  PROC DrawPart91()
    MoveL Offs(pOrigin,410.01,74.28,0.00),v60,z0,tPen\WObj:=wPaper;
    MoveL Offs(pOrigin,409.38,74.91,0.00),v40,z0,tPen\WObj:=wPaper;
    MoveL Offs(pOrigin,410.01,74.28,0.00),v40,fine,tPen\WObj:=wPaper;
    MoveL Offs(pOrigin,410.01,74.28,6.00),v60,z5,tPen\WObj:=wPaper;
    MoveL Offs(pOrigin,409.80,69.81,6.00),vTravel,z5,tPen\WObj:=wPaper;
    MoveL Offs(pOrigin,409.80,69.81,0.00),v60,z0,tPen\WObj:=wPaper;
    MoveL Offs(pOrigin,407.89,71.72,0.00),v40,z0,tPen\WObj:=wPaper;
    MoveL Offs(pOrigin,409.80,69.81,0.00),v40,fine,tPen\WObj:=wPaper;
    MoveL Offs(pOrigin,409.80,69.81,6.00),v60,z5,tPen\WObj:=wPaper;
    MoveL Offs(pOrigin,410.86,68.75,6.00),vTravel,z5,tPen\WObj:=wPaper;
    MoveL Offs(pOrigin,410.86,68.75,0.00),v60,z0,tPen\WObj:=wPaper;
    MoveL Offs(pOrigin,410.23,69.39,0.00),v40,z0,tPen\WObj:=wPaper;
    MoveL Offs(pOrigin,410.86,68.75,0.00),v40,fine,tPen\WObj:=wPaper;
    MoveL Offs(pOrigin,410.86,68.75,6.00),v60,z5,tPen\WObj:=wPaper;
    MoveL Offs(pOrigin,412.49,69.10,6.00),vTravel,z5,tPen\WObj:=wPaper;
    MoveL Offs(pOrigin,412.49,69.10,0.00),v60,z0,tPen\WObj:=wPaper;
    MoveL Offs(pOrigin,409.80,71.72,0.00),v40,z0,tPen\WObj:=wPaper;
    MoveL Offs(pOrigin,412.49,69.10,0.00),v40,fine,tPen\WObj:=wPaper;
    MoveL Offs(pOrigin,412.49,69.10,6.00),v60,z5,tPen\WObj:=wPaper;
    MoveL Offs(pOrigin,412.14,67.05,6.00),vTravel,z5,tPen\WObj:=wPaper;
    MoveL Offs(pOrigin,412.14,67.05,0.00),v60,z0,tPen\WObj:=wPaper;
    MoveL Offs(pOrigin,411.29,68.11,0.00),v40,z0,tPen\WObj:=wPaper;
    MoveL Offs(pOrigin,412.14,67.05,0.00),v40,fine,tPen\WObj:=wPaper;
    MoveL Offs(pOrigin,412.14,67.05,6.00),v60,z5,tPen\WObj:=wPaper;
    MoveL Offs(pOrigin,413.20,65.35,6.00),vTravel,z5,tPen\WObj:=wPaper;
    MoveL Offs(pOrigin,413.20,65.35,0.00),v60,z0,tPen\WObj:=wPaper;
    MoveL Offs(pOrigin,412.99,65.78,0.00),v40,z0,tPen\WObj:=wPaper;
    MoveL Offs(pOrigin,413.20,65.35,0.00),v40,fine,tPen\WObj:=wPaper;
    MoveL Offs(pOrigin,413.20,65.35,6.00),v60,z5,tPen\WObj:=wPaper;
    MoveL Offs(pOrigin,409.38,62.80,6.00),vTravel,z5,tPen\WObj:=wPaper;
    MoveL Offs(pOrigin,409.38,62.80,0.00),v60,z0,tPen\WObj:=wPaper;
    MoveL Offs(pOrigin,408.81,64.50,0.00),v40,z0,tPen\WObj:=wPaper;
    MoveL Offs(pOrigin,406.97,67.69,0.00),v40,z0,tPen\WObj:=wPaper;
    MoveL Offs(pOrigin,405.62,68.54,0.00),v40,z0,tPen\WObj:=wPaper;
    MoveL Offs(pOrigin,402.79,72.36,0.00),v40,z0,tPen\WObj:=wPaper;
    MoveL Offs(pOrigin,400.66,74.28,0.00),v40,fine,tPen\WObj:=wPaper;
    MoveL Offs(pOrigin,400.66,74.28,6.00),v60,z5,tPen\WObj:=wPaper;
    MoveL Offs(pOrigin,405.55,68.32,6.00),vTravel,z5,tPen\WObj:=wPaper;
    MoveL Offs(pOrigin,405.55,68.32,0.00),v60,z0,tPen\WObj:=wPaper;
    MoveL Offs(pOrigin,405.69,67.05,0.00),v40,z0,tPen\WObj:=wPaper;
    MoveL Offs(pOrigin,407.82,62.59,0.00),v40,z0,tPen\WObj:=wPaper;
    MoveL Offs(pOrigin,409.38,56.85,0.00),v40,z0,tPen\WObj:=wPaper;
    MoveL Offs(pOrigin,409.38,56.85,0.00),v40,z0,tPen\WObj:=wPaper;
    MoveL Offs(pOrigin,410.01,56.42,0.00),v40,z0,tPen\WObj:=wPaper;
    MoveL Offs(pOrigin,409.80,55.58,0.00),v40,z0,tPen\WObj:=wPaper;
    MoveL Offs(pOrigin,409.80,55.58,0.00),v40,z0,tPen\WObj:=wPaper;
    MoveL Offs(pOrigin,410.23,54.94,0.00),v40,z0,tPen\WObj:=wPaper;
    MoveL Offs(pOrigin,410.08,53.66,0.00),v40,z0,tPen\WObj:=wPaper;
    MoveL Offs(pOrigin,410.44,53.03,0.00),v40,z0,tPen\WObj:=wPaper;
    MoveL Offs(pOrigin,410.23,49.84,0.00),v40,z0,tPen\WObj:=wPaper;
    MoveL Offs(pOrigin,410.23,49.84,0.00),v40,z0,tPen\WObj:=wPaper;
    MoveL Offs(pOrigin,410.01,48.14,0.00),v40,z0,tPen\WObj:=wPaper;
    MoveL Offs(pOrigin,410.01,48.14,0.00),v40,z0,tPen\WObj:=wPaper;
    MoveL Offs(pOrigin,409.80,46.86,0.00),v40,z0,tPen\WObj:=wPaper;
    MoveL Offs(pOrigin,409.80,46.86,0.00),v40,z0,tPen\WObj:=wPaper;
    MoveL Offs(pOrigin,409.80,46.22,0.00),v40,z0,tPen\WObj:=wPaper;
    MoveL Offs(pOrigin,409.16,45.80,0.00),v40,z0,tPen\WObj:=wPaper;
    MoveL Offs(pOrigin,409.16,45.80,0.00),v40,z0,tPen\WObj:=wPaper;
    MoveL Offs(pOrigin,408.31,42.61,0.00),v40,fine,tPen\WObj:=wPaper;
    MoveL Offs(pOrigin,408.31,42.61,6.00),v60,z5,tPen\WObj:=wPaper;
    MoveL Offs(pOrigin,409.80,43.25,6.00),vTravel,z5,tPen\WObj:=wPaper;
    MoveL Offs(pOrigin,409.80,43.25,0.00),v60,z0,tPen\WObj:=wPaper;
    MoveL Offs(pOrigin,410.23,43.67,0.00),v40,z0,tPen\WObj:=wPaper;
    MoveL Offs(pOrigin,409.80,43.25,0.00),v40,fine,tPen\WObj:=wPaper;
    MoveL Offs(pOrigin,409.80,43.25,6.00),v60,z5,tPen\WObj:=wPaper;
    MoveL Offs(pOrigin,410.86,44.31,6.00),vTravel,z5,tPen\WObj:=wPaper;
    MoveL Offs(pOrigin,410.86,44.31,0.00),v60,z0,tPen\WObj:=wPaper;
    MoveL Offs(pOrigin,411.29,44.95,0.00),v40,z0,tPen\WObj:=wPaper;
    MoveL Offs(pOrigin,410.86,44.31,0.00),v40,fine,tPen\WObj:=wPaper;
    MoveL Offs(pOrigin,410.86,44.31,6.00),v60,z5,tPen\WObj:=wPaper;
    MoveL Offs(pOrigin,412.14,43.25,6.00),vTravel,z5,tPen\WObj:=wPaper;
    MoveL Offs(pOrigin,412.14,43.25,0.00),v60,z0,tPen\WObj:=wPaper;
    MoveL Offs(pOrigin,412.56,43.67,0.00),v40,z0,tPen\WObj:=wPaper;
    MoveL Offs(pOrigin,412.14,43.25,0.00),v40,fine,tPen\WObj:=wPaper;
    MoveL Offs(pOrigin,412.14,43.25,6.00),v60,z5,tPen\WObj:=wPaper;
    MoveL Offs(pOrigin,412.99,44.31,6.00),vTravel,z5,tPen\WObj:=wPaper;
    MoveL Offs(pOrigin,412.99,44.31,0.00),v60,z0,tPen\WObj:=wPaper;
    MoveL Offs(pOrigin,413.20,44.74,0.00),v40,z0,tPen\WObj:=wPaper;
    MoveL Offs(pOrigin,412.99,44.31,0.00),v40,z0,tPen\WObj:=wPaper;
    MoveL Offs(pOrigin,413.41,44.95,0.00),v40,z0,tPen\WObj:=wPaper;
    MoveL Offs(pOrigin,413.62,45.38,0.00),v40,z0,tPen\WObj:=wPaper;
    MoveL Offs(pOrigin,413.41,44.95,0.00),v40,z0,tPen\WObj:=wPaper;
    MoveL Offs(pOrigin,413.84,45.80,0.00),v40,z0,tPen\WObj:=wPaper;
    MoveL Offs(pOrigin,414.05,46.22,0.00),v40,z0,tPen\WObj:=wPaper;
    MoveL Offs(pOrigin,413.84,45.80,0.00),v40,fine,tPen\WObj:=wPaper;
    MoveL Offs(pOrigin,413.84,45.80,6.00),v60,z5,tPen\WObj:=wPaper;
    MoveL Offs(pOrigin,412.35,46.86,6.00),vTravel,z5,tPen\WObj:=wPaper;
    MoveL Offs(pOrigin,412.35,46.86,0.00),v60,z0,tPen\WObj:=wPaper;
    MoveL Offs(pOrigin,412.56,47.29,0.00),v40,z0,tPen\WObj:=wPaper;
    MoveL Offs(pOrigin,412.35,46.86,0.00),v40,fine,tPen\WObj:=wPaper;
    MoveL Offs(pOrigin,412.35,46.86,6.00),v60,z5,tPen\WObj:=wPaper;
    MoveL Offs(pOrigin,409.16,46.86,6.00),vTravel,z5,tPen\WObj:=wPaper;
    MoveL Offs(pOrigin,409.16,46.86,0.00),v60,z0,tPen\WObj:=wPaper;
    MoveL Offs(pOrigin,408.95,46.01,0.00),v40,z0,tPen\WObj:=wPaper;
    MoveL Offs(pOrigin,409.16,45.80,0.00),v40,z0,tPen\WObj:=wPaper;
    MoveL Offs(pOrigin,409.16,46.86,0.00),v40,z0,tPen\WObj:=wPaper;
    MoveL Offs(pOrigin,409.38,48.14,0.00),v40,z0,tPen\WObj:=wPaper;
    MoveL Offs(pOrigin,409.38,48.14,0.00),v40,z0,tPen\WObj:=wPaper;
    MoveL Offs(pOrigin,409.59,49.84,0.00),v40,z0,tPen\WObj:=wPaper;
    MoveL Offs(pOrigin,409.59,49.84,0.00),v40,z0,tPen\WObj:=wPaper;
    MoveL Offs(pOrigin,409.80,53.66,0.00),v40,z0,tPen\WObj:=wPaper;
    MoveL Offs(pOrigin,410.01,54.09,0.00),v40,z0,tPen\WObj:=wPaper;
    MoveL Offs(pOrigin,409.80,53.88,0.00),v40,z0,tPen\WObj:=wPaper;
    MoveL Offs(pOrigin,409.38,54.30,0.00),v40,z0,tPen\WObj:=wPaper;
    MoveL Offs(pOrigin,409.38,55.36,0.00),v40,z0,tPen\WObj:=wPaper;
    MoveL Offs(pOrigin,409.80,55.58,0.00),v40,z0,tPen\WObj:=wPaper;
    MoveL Offs(pOrigin,409.38,55.58,0.00),v40,z0,tPen\WObj:=wPaper;
    MoveL Offs(pOrigin,409.16,56.64,0.00),v40,z0,tPen\WObj:=wPaper;
    MoveL Offs(pOrigin,409.38,56.85,0.00),v40,fine,tPen\WObj:=wPaper;
    MoveL Offs(pOrigin,409.38,56.85,6.00),v60,z5,tPen\WObj:=wPaper;
    MoveL Offs(pOrigin,407.04,64.07,6.00),vTravel,z5,tPen\WObj:=wPaper;
    MoveL Offs(pOrigin,407.04,64.07,0.00),v60,z0,tPen\WObj:=wPaper;
    MoveL Offs(pOrigin,406.83,64.50,0.00),v40,z0,tPen\WObj:=wPaper;
    MoveL Offs(pOrigin,407.04,64.07,0.00),v40,fine,tPen\WObj:=wPaper;
    MoveL Offs(pOrigin,407.04,64.07,6.00),v60,z5,tPen\WObj:=wPaper;
    MoveL Offs(pOrigin,397.69,57.49,6.00),vTravel,z5,tPen\WObj:=wPaper;
    MoveL Offs(pOrigin,397.69,57.49,0.00),v60,z0,tPen\WObj:=wPaper;
    MoveL Offs(pOrigin,397.26,58.12,0.00),v40,z0,tPen\WObj:=wPaper;
    MoveL Offs(pOrigin,397.69,57.49,0.00),v40,fine,tPen\WObj:=wPaper;
    MoveL Offs(pOrigin,397.69,57.49,6.00),v60,z5,tPen\WObj:=wPaper;
  ENDPROC

  PROC DrawPart92()
    MoveL Offs(pOrigin,398.33,56.42,6.00),vTravel,z5,tPen\WObj:=wPaper;
    MoveL Offs(pOrigin,398.33,56.42,0.00),v60,z0,tPen\WObj:=wPaper;
    MoveL Offs(pOrigin,398.11,56.85,0.00),v40,z0,tPen\WObj:=wPaper;
    MoveL Offs(pOrigin,398.33,56.42,0.00),v40,fine,tPen\WObj:=wPaper;
    MoveL Offs(pOrigin,398.33,56.42,6.00),v60,z5,tPen\WObj:=wPaper;
    MoveL Offs(pOrigin,396.84,58.76,6.00),vTravel,z5,tPen\WObj:=wPaper;
    MoveL Offs(pOrigin,396.84,58.76,0.00),v60,z0,tPen\WObj:=wPaper;
    MoveL Offs(pOrigin,396.41,59.40,0.00),v40,z0,tPen\WObj:=wPaper;
    MoveL Offs(pOrigin,396.84,58.76,0.00),v40,fine,tPen\WObj:=wPaper;
    MoveL Offs(pOrigin,396.84,58.76,6.00),v60,z5,tPen\WObj:=wPaper;
    MoveL Offs(pOrigin,395.56,60.67,6.00),vTravel,z5,tPen\WObj:=wPaper;
    MoveL Offs(pOrigin,395.56,60.67,0.00),v60,z0,tPen\WObj:=wPaper;
    MoveL Offs(pOrigin,395.14,61.10,0.00),v40,z0,tPen\WObj:=wPaper;
    MoveL Offs(pOrigin,395.56,60.67,0.00),v40,fine,tPen\WObj:=wPaper;
    MoveL Offs(pOrigin,395.56,60.67,6.00),v60,z5,tPen\WObj:=wPaper;
    MoveL Offs(pOrigin,394.29,62.16,6.00),vTravel,z5,tPen\WObj:=wPaper;
    MoveL Offs(pOrigin,394.29,62.16,0.00),v60,z0,tPen\WObj:=wPaper;
    MoveL Offs(pOrigin,393.86,62.80,0.00),v40,z0,tPen\WObj:=wPaper;
    MoveL Offs(pOrigin,394.29,62.16,0.00),v40,fine,tPen\WObj:=wPaper;
    MoveL Offs(pOrigin,394.29,62.16,6.00),v60,z5,tPen\WObj:=wPaper;
    MoveL Offs(pOrigin,393.44,63.22,6.00),vTravel,z5,tPen\WObj:=wPaper;
    MoveL Offs(pOrigin,393.44,63.22,0.00),v60,z0,tPen\WObj:=wPaper;
    MoveL Offs(pOrigin,393.01,63.65,0.00),v40,z0,tPen\WObj:=wPaper;
    MoveL Offs(pOrigin,393.44,63.22,0.00),v40,fine,tPen\WObj:=wPaper;
    MoveL Offs(pOrigin,393.44,63.22,6.00),v60,z5,tPen\WObj:=wPaper;
    MoveL Offs(pOrigin,392.16,64.71,6.00),vTravel,z5,tPen\WObj:=wPaper;
    MoveL Offs(pOrigin,392.16,64.71,0.00),v60,z0,tPen\WObj:=wPaper;
    MoveL Offs(pOrigin,391.52,65.35,0.00),v40,z0,tPen\WObj:=wPaper;
    MoveL Offs(pOrigin,392.16,64.71,0.00),v40,fine,tPen\WObj:=wPaper;
    MoveL Offs(pOrigin,392.16,64.71,6.00),v60,z5,tPen\WObj:=wPaper;
    MoveL Offs(pOrigin,391.31,65.56,6.00),vTravel,z5,tPen\WObj:=wPaper;
    MoveL Offs(pOrigin,391.31,65.56,0.00),v60,z0,tPen\WObj:=wPaper;
    MoveL Offs(pOrigin,390.67,66.20,0.00),v40,z0,tPen\WObj:=wPaper;
    MoveL Offs(pOrigin,391.31,65.56,0.00),v40,fine,tPen\WObj:=wPaper;
    MoveL Offs(pOrigin,391.31,65.56,6.00),v60,z5,tPen\WObj:=wPaper;
    MoveL Offs(pOrigin,389.61,67.05,6.00),vTravel,z5,tPen\WObj:=wPaper;
    MoveL Offs(pOrigin,389.61,67.05,0.00),v60,z0,tPen\WObj:=wPaper;
    MoveL Offs(pOrigin,388.98,67.69,0.00),v40,z0,tPen\WObj:=wPaper;
    MoveL Offs(pOrigin,389.61,67.05,0.00),v40,fine,tPen\WObj:=wPaper;
    MoveL Offs(pOrigin,389.61,67.05,6.00),v60,z5,tPen\WObj:=wPaper;
    MoveL Offs(pOrigin,399.81,53.66,6.00),vTravel,z5,tPen\WObj:=wPaper;
    MoveL Offs(pOrigin,399.81,53.66,0.00),v60,z0,tPen\WObj:=wPaper;
    MoveL Offs(pOrigin,399.60,54.09,0.00),v40,z0,tPen\WObj:=wPaper;
    MoveL Offs(pOrigin,399.81,53.66,0.00),v40,fine,tPen\WObj:=wPaper;
    MoveL Offs(pOrigin,399.81,53.66,6.00),v60,z5,tPen\WObj:=wPaper;
    MoveL Offs(pOrigin,402.58,42.19,6.00),vTravel,z5,tPen\WObj:=wPaper;
    MoveL Offs(pOrigin,402.58,42.19,0.00),v60,z0,tPen\WObj:=wPaper;
    MoveL Offs(pOrigin,401.94,47.71,0.00),v40,z0,tPen\WObj:=wPaper;
    MoveL Offs(pOrigin,399.88,53.88,0.00),v40,z0,tPen\WObj:=wPaper;
    MoveL Offs(pOrigin,396.20,60.04,0.00),v40,z0,tPen\WObj:=wPaper;
    MoveL Offs(pOrigin,392.59,64.50,0.00),v40,z0,tPen\WObj:=wPaper;
    MoveL Offs(pOrigin,387.91,68.75,0.00),v40,z0,tPen\WObj:=wPaper;
    MoveL Offs(pOrigin,382.81,72.22,0.00),v40,z0,tPen\WObj:=wPaper;
    MoveL Offs(pOrigin,377.08,74.77,0.00),v40,z0,tPen\WObj:=wPaper;
    MoveL Offs(pOrigin,370.49,76.40,0.00),v40,z0,tPen\WObj:=wPaper;
    MoveL Offs(pOrigin,370.42,76.19,0.00),v40,z0,tPen\WObj:=wPaper;
    MoveL Offs(pOrigin,369.64,75.97,0.00),v40,z0,tPen\WObj:=wPaper;
    MoveL Offs(pOrigin,369.00,76.61,0.00),v40,z0,tPen\WObj:=wPaper;
    MoveL Offs(pOrigin,369.85,76.82,0.00),v40,z0,tPen\WObj:=wPaper;
    MoveL Offs(pOrigin,370.42,76.19,0.00),v40,fine,tPen\WObj:=wPaper;
    MoveL Offs(pOrigin,370.42,76.19,6.00),v60,z5,tPen\WObj:=wPaper;
    MoveL Offs(pOrigin,381.96,113.38,6.00),vTravel,z5,tPen\WObj:=wPaper;
    MoveL Offs(pOrigin,381.96,113.38,0.00),v60,z0,tPen\WObj:=wPaper;
    MoveL Offs(pOrigin,386.42,112.74,0.00),v40,z0,tPen\WObj:=wPaper;
    MoveL Offs(pOrigin,391.10,111.46,0.00),v40,z0,tPen\WObj:=wPaper;
    MoveL Offs(pOrigin,391.10,111.46,0.00),v40,z0,tPen\WObj:=wPaper;
    MoveL Offs(pOrigin,393.86,110.68,0.00),v40,z0,tPen\WObj:=wPaper;
    MoveL Offs(pOrigin,399.17,107.71,0.00),v40,z0,tPen\WObj:=wPaper;
    MoveL Offs(pOrigin,399.95,107.64,0.00),v40,z0,tPen\WObj:=wPaper;
    MoveL Offs(pOrigin,400.02,108.28,0.00),v40,z0,tPen\WObj:=wPaper;
    MoveL Offs(pOrigin,398.61,112.53,0.00),v40,z0,tPen\WObj:=wPaper;
    MoveL Offs(pOrigin,396.06,116.21,0.00),v40,z0,tPen\WObj:=wPaper;
    MoveL Offs(pOrigin,395.14,118.47,0.00),v40,z0,tPen\WObj:=wPaper;
    MoveL Offs(pOrigin,395.35,125.06,0.00),v40,z0,tPen\WObj:=wPaper;
    MoveL Offs(pOrigin,395.00,126.12,0.00),v40,z0,tPen\WObj:=wPaper;
    MoveL Offs(pOrigin,393.65,126.97,0.00),v40,z0,tPen\WObj:=wPaper;
    MoveL Offs(pOrigin,392.16,126.97,0.00),v40,z0,tPen\WObj:=wPaper;
    MoveL Offs(pOrigin,385.36,125.49,0.00),v40,z0,tPen\WObj:=wPaper;
    MoveL Offs(pOrigin,384.51,125.70,0.00),v40,z0,tPen\WObj:=wPaper;
    MoveL Offs(pOrigin,384.51,125.70,0.00),v40,z0,tPen\WObj:=wPaper;
    MoveL Offs(pOrigin,378.99,124.64,0.00),v40,fine,tPen\WObj:=wPaper;
    MoveL Offs(pOrigin,378.99,124.64,6.00),v60,z5,tPen\WObj:=wPaper;
    MoveL Offs(pOrigin,394.71,126.34,6.00),vTravel,z5,tPen\WObj:=wPaper;
    MoveL Offs(pOrigin,394.71,126.34,0.00),v60,z0,tPen\WObj:=wPaper;
    MoveL Offs(pOrigin,394.50,126.76,0.00),v40,z0,tPen\WObj:=wPaper;
    MoveL Offs(pOrigin,394.71,126.34,0.00),v40,fine,tPen\WObj:=wPaper;
    MoveL Offs(pOrigin,394.71,126.34,6.00),v60,z5,tPen\WObj:=wPaper;
    MoveL Offs(pOrigin,396.41,126.55,6.00),vTravel,z5,tPen\WObj:=wPaper;
    MoveL Offs(pOrigin,396.41,126.55,0.00),v60,z0,tPen\WObj:=wPaper;
    MoveL Offs(pOrigin,396.20,126.97,0.00),v40,z0,tPen\WObj:=wPaper;
    MoveL Offs(pOrigin,396.41,126.55,0.00),v40,fine,tPen\WObj:=wPaper;
    MoveL Offs(pOrigin,396.41,126.55,6.00),v60,z5,tPen\WObj:=wPaper;
    MoveL Offs(pOrigin,397.26,117.20,6.00),vTravel,z5,tPen\WObj:=wPaper;
    MoveL Offs(pOrigin,397.26,117.20,0.00),v60,z0,tPen\WObj:=wPaper;
    MoveL Offs(pOrigin,397.05,117.62,0.00),v40,z0,tPen\WObj:=wPaper;
    MoveL Offs(pOrigin,397.26,117.20,0.00),v40,fine,tPen\WObj:=wPaper;
    MoveL Offs(pOrigin,397.26,117.20,6.00),v60,z5,tPen\WObj:=wPaper;
    MoveL Offs(pOrigin,398.11,116.14,6.00),vTravel,z5,tPen\WObj:=wPaper;
    MoveL Offs(pOrigin,398.11,116.14,0.00),v60,z0,tPen\WObj:=wPaper;
    MoveL Offs(pOrigin,398.33,115.71,0.00),v40,z0,tPen\WObj:=wPaper;
    MoveL Offs(pOrigin,398.11,116.14,0.00),v40,fine,tPen\WObj:=wPaper;
    MoveL Offs(pOrigin,398.11,116.14,6.00),v60,z5,tPen\WObj:=wPaper;
    MoveL Offs(pOrigin,396.84,115.07,6.00),vTravel,z5,tPen\WObj:=wPaper;
    MoveL Offs(pOrigin,396.84,115.07,0.00),v60,z0,tPen\WObj:=wPaper;
    MoveL Offs(pOrigin,396.62,115.50,0.00),v40,z0,tPen\WObj:=wPaper;
    MoveL Offs(pOrigin,396.84,115.07,0.00),v40,fine,tPen\WObj:=wPaper;
    MoveL Offs(pOrigin,396.84,115.07,6.00),v60,z5,tPen\WObj:=wPaper;
    MoveL Offs(pOrigin,399.81,113.38,6.00),vTravel,z5,tPen\WObj:=wPaper;
    MoveL Offs(pOrigin,399.81,113.38,0.00),v60,z0,tPen\WObj:=wPaper;
    MoveL Offs(pOrigin,399.60,113.80,0.00),v40,z0,tPen\WObj:=wPaper;
    MoveL Offs(pOrigin,399.81,113.38,0.00),v40,fine,tPen\WObj:=wPaper;
    MoveL Offs(pOrigin,399.81,113.38,6.00),v60,z5,tPen\WObj:=wPaper;
    MoveL Offs(pOrigin,398.11,106.79,6.00),vTravel,z5,tPen\WObj:=wPaper;
    MoveL Offs(pOrigin,398.11,106.79,0.00),v60,z0,tPen\WObj:=wPaper;
    MoveL Offs(pOrigin,398.40,106.65,0.00),v40,z0,tPen\WObj:=wPaper;
    MoveL Offs(pOrigin,395.35,108.77,0.00),v40,z0,tPen\WObj:=wPaper;
    MoveL Offs(pOrigin,391.74,110.54,0.00),v40,z0,tPen\WObj:=wPaper;
    MoveL Offs(pOrigin,391.10,111.46,0.00),v40,fine,tPen\WObj:=wPaper;
    MoveL Offs(pOrigin,391.10,111.46,6.00),v60,z5,tPen\WObj:=wPaper;
    MoveL Offs(pOrigin,403.21,104.24,6.00),vTravel,z5,tPen\WObj:=wPaper;
  ENDPROC

  PROC DrawPart93()
    MoveL Offs(pOrigin,403.21,104.24,0.00),v60,z0,tPen\WObj:=wPaper;
    MoveL Offs(pOrigin,403.00,104.66,0.00),v40,z0,tPen\WObj:=wPaper;
    MoveL Offs(pOrigin,403.21,104.24,0.00),v40,z0,tPen\WObj:=wPaper;
    MoveL Offs(pOrigin,403.85,103.60,0.00),v40,z0,tPen\WObj:=wPaper;
    MoveL Offs(pOrigin,403.64,104.03,0.00),v40,z0,tPen\WObj:=wPaper;
    MoveL Offs(pOrigin,403.85,103.60,0.00),v40,fine,tPen\WObj:=wPaper;
    MoveL Offs(pOrigin,403.85,103.60,6.00),v60,z5,tPen\WObj:=wPaper;
    MoveL Offs(pOrigin,385.58,153.32,6.00),vTravel,z5,tPen\WObj:=wPaper;
    MoveL Offs(pOrigin,385.58,153.32,0.00),v60,z0,tPen\WObj:=wPaper;
    MoveL Offs(pOrigin,385.36,153.75,0.00),v40,z0,tPen\WObj:=wPaper;
    MoveL Offs(pOrigin,385.58,153.32,0.00),v40,fine,tPen\WObj:=wPaper;
    MoveL Offs(pOrigin,385.58,153.32,6.00),v60,z5,tPen\WObj:=wPaper;
    MoveL Offs(pOrigin,383.88,153.11,6.00),vTravel,z5,tPen\WObj:=wPaper;
    MoveL Offs(pOrigin,383.88,153.11,0.00),v60,z0,tPen\WObj:=wPaper;
    MoveL Offs(pOrigin,383.66,153.54,0.00),v40,z0,tPen\WObj:=wPaper;
    MoveL Offs(pOrigin,383.88,153.11,0.00),v40,fine,tPen\WObj:=wPaper;
    MoveL Offs(pOrigin,383.88,153.11,6.00),v60,z5,tPen\WObj:=wPaper;
    MoveL Offs(pOrigin,383.24,154.60,6.00),vTravel,z5,tPen\WObj:=wPaper;
    MoveL Offs(pOrigin,383.24,154.60,0.00),v60,z0,tPen\WObj:=wPaper;
    MoveL Offs(pOrigin,383.02,155.02,0.00),v40,z0,tPen\WObj:=wPaper;
    MoveL Offs(pOrigin,383.24,154.60,0.00),v40,z0,tPen\WObj:=wPaper;
    MoveL Offs(pOrigin,382.81,155.45,0.00),v40,z0,tPen\WObj:=wPaper;
    MoveL Offs(pOrigin,382.60,155.88,0.00),v40,z0,tPen\WObj:=wPaper;
    MoveL Offs(pOrigin,382.81,155.45,0.00),v40,z0,tPen\WObj:=wPaper;
    MoveL Offs(pOrigin,382.39,156.30,0.00),v40,z0,tPen\WObj:=wPaper;
    MoveL Offs(pOrigin,382.17,156.73,0.00),v40,z0,tPen\WObj:=wPaper;
    MoveL Offs(pOrigin,382.39,156.30,0.00),v40,fine,tPen\WObj:=wPaper;
    MoveL Offs(pOrigin,382.39,156.30,6.00),v60,z5,tPen\WObj:=wPaper;
    MoveL Offs(pOrigin,381.75,157.57,6.00),vTravel,z5,tPen\WObj:=wPaper;
    MoveL Offs(pOrigin,381.75,157.57,0.00),v60,z0,tPen\WObj:=wPaper;
    MoveL Offs(pOrigin,381.54,158.00,0.00),v40,z0,tPen\WObj:=wPaper;
    MoveL Offs(pOrigin,381.75,157.57,0.00),v40,fine,tPen\WObj:=wPaper;
    MoveL Offs(pOrigin,381.75,157.57,6.00),v60,z5,tPen\WObj:=wPaper;
    MoveL Offs(pOrigin,383.02,158.64,6.00),vTravel,z5,tPen\WObj:=wPaper;
    MoveL Offs(pOrigin,383.02,158.64,0.00),v60,z0,tPen\WObj:=wPaper;
    MoveL Offs(pOrigin,382.81,159.06,0.00),v40,z0,tPen\WObj:=wPaper;
    MoveL Offs(pOrigin,383.02,158.64,0.00),v40,z0,tPen\WObj:=wPaper;
    MoveL Offs(pOrigin,383.45,157.79,0.00),v40,z0,tPen\WObj:=wPaper;
    MoveL Offs(pOrigin,383.24,158.21,0.00),v40,z0,tPen\WObj:=wPaper;
    MoveL Offs(pOrigin,383.45,157.79,0.00),v40,fine,tPen\WObj:=wPaper;
    MoveL Offs(pOrigin,383.45,157.79,6.00),v60,z5,tPen\WObj:=wPaper;
    MoveL Offs(pOrigin,384.51,155.66,6.00),vTravel,z5,tPen\WObj:=wPaper;
    MoveL Offs(pOrigin,384.51,155.66,0.00),v60,z0,tPen\WObj:=wPaper;
    MoveL Offs(pOrigin,384.30,156.09,0.00),v40,z0,tPen\WObj:=wPaper;
    MoveL Offs(pOrigin,384.51,155.66,0.00),v40,fine,tPen\WObj:=wPaper;
    MoveL Offs(pOrigin,384.51,155.66,6.00),v60,z5,tPen\WObj:=wPaper;
    MoveL Offs(pOrigin,369.42,186.48,6.00),vTravel,z5,tPen\WObj:=wPaper;
    MoveL Offs(pOrigin,369.42,186.48,0.00),v60,z0,tPen\WObj:=wPaper;
    MoveL Offs(pOrigin,369.64,186.90,0.00),v40,z0,tPen\WObj:=wPaper;
    MoveL Offs(pOrigin,369.42,186.48,0.00),v40,fine,tPen\WObj:=wPaper;
    MoveL Offs(pOrigin,369.42,186.48,6.00),v60,z5,tPen\WObj:=wPaper;
    MoveL Offs(pOrigin,368.58,187.75,6.00),vTravel,z5,tPen\WObj:=wPaper;
    MoveL Offs(pOrigin,368.58,187.75,0.00),v60,z0,tPen\WObj:=wPaper;
    MoveL Offs(pOrigin,369.00,188.18,0.00),v40,z0,tPen\WObj:=wPaper;
    MoveL Offs(pOrigin,368.58,187.75,0.00),v40,fine,tPen\WObj:=wPaper;
    MoveL Offs(pOrigin,368.58,187.75,6.00),v60,z5,tPen\WObj:=wPaper;
    MoveL Offs(pOrigin,367.73,186.26,6.00),vTravel,z5,tPen\WObj:=wPaper;
    MoveL Offs(pOrigin,367.73,186.26,0.00),v60,z0,tPen\WObj:=wPaper;
    MoveL Offs(pOrigin,367.94,186.69,0.00),v40,z0,tPen\WObj:=wPaper;
    MoveL Offs(pOrigin,367.73,186.26,0.00),v40,fine,tPen\WObj:=wPaper;
    MoveL Offs(pOrigin,367.73,186.26,6.00),v60,z5,tPen\WObj:=wPaper;
    MoveL Offs(pOrigin,341.80,182.01,6.00),vTravel,z5,tPen\WObj:=wPaper;
    MoveL Offs(pOrigin,341.80,182.01,0.00),v60,z0,tPen\WObj:=wPaper;
    MoveL Offs(pOrigin,334.15,175.85,0.00),v40,z0,tPen\WObj:=wPaper;
    MoveL Offs(pOrigin,330.33,172.02,0.00),v40,z0,tPen\WObj:=wPaper;
    MoveL Offs(pOrigin,323.74,164.16,0.00),v40,z0,tPen\WObj:=wPaper;
    MoveL Offs(pOrigin,315.38,151.84,0.00),v40,z0,tPen\WObj:=wPaper;
    MoveL Offs(pOrigin,309.85,141.64,0.00),v40,z0,tPen\WObj:=wPaper;
    MoveL Offs(pOrigin,309.08,139.51,0.00),v40,fine,tPen\WObj:=wPaper;
    MoveL Offs(pOrigin,309.08,139.51,6.00),v60,z5,tPen\WObj:=wPaper;
    MoveL Offs(pOrigin,316.73,153.75,6.00),vTravel,z5,tPen\WObj:=wPaper;
    MoveL Offs(pOrigin,316.73,153.75,0.00),v60,z0,tPen\WObj:=wPaper;
    MoveL Offs(pOrigin,316.94,154.18,0.00),v40,z0,tPen\WObj:=wPaper;
    MoveL Offs(pOrigin,316.73,153.75,0.00),v40,z0,tPen\WObj:=wPaper;
    MoveL Offs(pOrigin,317.15,154.39,0.00),v40,z0,tPen\WObj:=wPaper;
    MoveL Offs(pOrigin,317.36,154.81,0.00),v40,z0,tPen\WObj:=wPaper;
    MoveL Offs(pOrigin,317.15,154.39,0.00),v40,fine,tPen\WObj:=wPaper;
    MoveL Offs(pOrigin,317.15,154.39,6.00),v60,z5,tPen\WObj:=wPaper;
    MoveL Offs(pOrigin,305.25,169.69,6.00),vTravel,z5,tPen\WObj:=wPaper;
    MoveL Offs(pOrigin,305.25,169.69,0.00),v60,z0,tPen\WObj:=wPaper;
    MoveL Offs(pOrigin,295.90,173.09,0.00),v40,fine,tPen\WObj:=wPaper;
    MoveL Offs(pOrigin,295.90,173.09,6.00),v60,z5,tPen\WObj:=wPaper;
    MoveL Offs(pOrigin,276.56,176.70,6.00),vTravel,z5,tPen\WObj:=wPaper;
    MoveL Offs(pOrigin,276.56,176.70,0.00),v60,z0,tPen\WObj:=wPaper;
    MoveL Offs(pOrigin,276.00,174.36,0.00),v40,z0,tPen\WObj:=wPaper;
    MoveL Offs(pOrigin,271.82,165.44,0.00),v40,z0,tPen\WObj:=wPaper;
    MoveL Offs(pOrigin,268.70,157.15,0.00),v40,fine,tPen\WObj:=wPaper;
    MoveL Offs(pOrigin,268.70,157.15,6.00),v60,z5,tPen\WObj:=wPaper;
    MoveL Offs(pOrigin,274.44,150.56,6.00),vTravel,z5,tPen\WObj:=wPaper;
    MoveL Offs(pOrigin,274.44,150.56,0.00),v60,z0,tPen\WObj:=wPaper;
    MoveL Offs(pOrigin,273.73,149.93,0.00),v40,z0,tPen\WObj:=wPaper;
    MoveL Offs(pOrigin,267.78,135.05,0.00),v40,z0,tPen\WObj:=wPaper;
    MoveL Offs(pOrigin,267.64,133.77,0.00),v40,fine,tPen\WObj:=wPaper;
    MoveL Offs(pOrigin,267.64,133.77,6.00),v60,z5,tPen\WObj:=wPaper;
    MoveL Offs(pOrigin,276.14,186.48,6.00),vTravel,z5,tPen\WObj:=wPaper;
    MoveL Offs(pOrigin,276.14,186.48,0.00),v60,z0,tPen\WObj:=wPaper;
    MoveL Offs(pOrigin,275.71,187.11,0.00),v40,z0,tPen\WObj:=wPaper;
    MoveL Offs(pOrigin,276.14,186.48,0.00),v40,fine,tPen\WObj:=wPaper;
    MoveL Offs(pOrigin,276.14,186.48,6.00),v60,z5,tPen\WObj:=wPaper;
    MoveL Offs(pOrigin,303.55,208.15,6.00),vTravel,z5,tPen\WObj:=wPaper;
    MoveL Offs(pOrigin,303.55,208.15,0.00),v60,z0,tPen\WObj:=wPaper;
    MoveL Offs(pOrigin,303.12,208.79,0.00),v40,z0,tPen\WObj:=wPaper;
    MoveL Offs(pOrigin,303.55,208.15,0.00),v40,fine,tPen\WObj:=wPaper;
    MoveL Offs(pOrigin,303.55,208.15,6.00),v60,z5,tPen\WObj:=wPaper;
    MoveL Offs(pOrigin,304.40,207.30,6.00),vTravel,z5,tPen\WObj:=wPaper;
    MoveL Offs(pOrigin,304.40,207.30,0.00),v60,z0,tPen\WObj:=wPaper;
    MoveL Offs(pOrigin,303.76,207.94,0.00),v40,z0,tPen\WObj:=wPaper;
    MoveL Offs(pOrigin,304.40,207.30,0.00),v40,fine,tPen\WObj:=wPaper;
    MoveL Offs(pOrigin,304.40,207.30,6.00),v60,z5,tPen\WObj:=wPaper;
    MoveL Offs(pOrigin,314.60,193.91,6.00),vTravel,z5,tPen\WObj:=wPaper;
    MoveL Offs(pOrigin,314.60,193.91,0.00),v60,z0,tPen\WObj:=wPaper;
    MoveL Offs(pOrigin,315.02,194.12,0.00),v40,z0,tPen\WObj:=wPaper;
    MoveL Offs(pOrigin,314.60,193.91,0.00),v40,fine,tPen\WObj:=wPaper;
    MoveL Offs(pOrigin,314.60,193.91,6.00),v60,z5,tPen\WObj:=wPaper;
    MoveL Offs(pOrigin,332.66,174.15,6.00),vTravel,z5,tPen\WObj:=wPaper;
    MoveL Offs(pOrigin,332.66,174.15,0.00),v60,z0,tPen\WObj:=wPaper;
    MoveL Offs(pOrigin,333.51,175.00,0.00),v40,z0,tPen\WObj:=wPaper;
    MoveL Offs(pOrigin,332.66,174.15,0.00),v40,fine,tPen\WObj:=wPaper;
    MoveL Offs(pOrigin,332.66,174.15,6.00),v60,z5,tPen\WObj:=wPaper;
    MoveL Offs(pOrigin,331.17,172.66,6.00),vTravel,z5,tPen\WObj:=wPaper;
  ENDPROC

  PROC DrawPart94()
    MoveL Offs(pOrigin,331.17,172.66,0.00),v60,z0,tPen\WObj:=wPaper;
    MoveL Offs(pOrigin,332.02,173.51,0.00),v40,z0,tPen\WObj:=wPaper;
    MoveL Offs(pOrigin,331.17,172.66,0.00),v40,fine,tPen\WObj:=wPaper;
    MoveL Offs(pOrigin,331.17,172.66,6.00),v60,z5,tPen\WObj:=wPaper;
    MoveL Offs(pOrigin,383.66,227.27,6.00),vTravel,z5,tPen\WObj:=wPaper;
    MoveL Offs(pOrigin,383.66,227.27,0.00),v60,z0,tPen\WObj:=wPaper;
    MoveL Offs(pOrigin,383.45,227.70,0.00),v40,z0,tPen\WObj:=wPaper;
    MoveL Offs(pOrigin,383.66,227.27,0.00),v40,fine,tPen\WObj:=wPaper;
    MoveL Offs(pOrigin,383.66,227.27,6.00),v60,z5,tPen\WObj:=wPaper;
    MoveL Offs(pOrigin,250.85,225.57,6.00),vTravel,z5,tPen\WObj:=wPaper;
    MoveL Offs(pOrigin,250.85,225.57,0.00),v60,z0,tPen\WObj:=wPaper;
    MoveL Offs(pOrigin,245.54,225.15,0.00),v40,z0,tPen\WObj:=wPaper;
    MoveL Offs(pOrigin,242.56,224.30,0.00),v40,fine,tPen\WObj:=wPaper;
    MoveL Offs(pOrigin,242.56,224.30,6.00),v60,z5,tPen\WObj:=wPaper;
    MoveL Offs(pOrigin,232.15,237.05,6.00),vTravel,z5,tPen\WObj:=wPaper;
    MoveL Offs(pOrigin,232.15,237.05,0.00),v60,z0,tPen\WObj:=wPaper;
    MoveL Offs(pOrigin,232.57,237.26,0.00),v40,z0,tPen\WObj:=wPaper;
    MoveL Offs(pOrigin,232.57,238.11,0.00),v40,z0,tPen\WObj:=wPaper;
    MoveL Offs(pOrigin,231.73,238.11,0.00),v40,z0,tPen\WObj:=wPaper;
    MoveL Offs(pOrigin,231.94,238.96,0.00),v40,z0,tPen\WObj:=wPaper;
    MoveL Offs(pOrigin,233.00,239.18,0.00),v40,z0,tPen\WObj:=wPaper;
    MoveL Offs(pOrigin,233.43,238.75,0.00),v40,z0,tPen\WObj:=wPaper;
    MoveL Offs(pOrigin,233.43,238.11,0.00),v40,z0,tPen\WObj:=wPaper;
    MoveL Offs(pOrigin,233.64,238.68,0.00),v40,z0,tPen\WObj:=wPaper;
    MoveL Offs(pOrigin,235.34,239.39,0.00),v40,z0,tPen\WObj:=wPaper;
    MoveL Offs(pOrigin,235.76,240.45,0.00),v40,z0,tPen\WObj:=wPaper;
    MoveL Offs(pOrigin,235.76,240.45,0.00),v40,z0,tPen\WObj:=wPaper;
    MoveL Offs(pOrigin,234.70,240.88,0.00),v40,z0,tPen\WObj:=wPaper;
    MoveL Offs(pOrigin,234.49,241.51,0.00),v40,fine,tPen\WObj:=wPaper;
    MoveL Offs(pOrigin,234.49,241.51,6.00),v60,z5,tPen\WObj:=wPaper;
    MoveL Offs(pOrigin,238.10,242.36,6.00),vTravel,z5,tPen\WObj:=wPaper;
    MoveL Offs(pOrigin,238.10,242.36,0.00),v60,z0,tPen\WObj:=wPaper;
    MoveL Offs(pOrigin,238.31,241.94,0.00),v40,z0,tPen\WObj:=wPaper;
    MoveL Offs(pOrigin,239.16,241.73,0.00),v40,fine,tPen\WObj:=wPaper;
    MoveL Offs(pOrigin,239.16,241.73,6.00),v60,z5,tPen\WObj:=wPaper;
    MoveL Offs(pOrigin,238.10,242.36,6.00),vTravel,z5,tPen\WObj:=wPaper;
    MoveL Offs(pOrigin,238.10,242.36,0.00),v60,z0,tPen\WObj:=wPaper;
    MoveL Offs(pOrigin,236.19,242.57,0.00),v40,z0,tPen\WObj:=wPaper;
    MoveL Offs(pOrigin,233.85,241.58,0.00),v40,z0,tPen\WObj:=wPaper;
    MoveL Offs(pOrigin,232.43,243.00,0.00),v40,z0,tPen\WObj:=wPaper;
    MoveL Offs(pOrigin,231.73,246.19,0.00),v40,fine,tPen\WObj:=wPaper;
    MoveL Offs(pOrigin,231.73,246.19,6.00),v60,z5,tPen\WObj:=wPaper;
    MoveL Offs(pOrigin,231.09,237.90,6.00),vTravel,z5,tPen\WObj:=wPaper;
    MoveL Offs(pOrigin,231.09,237.90,0.00),v60,z0,tPen\WObj:=wPaper;
    MoveL Offs(pOrigin,232.15,237.05,0.00),v40,fine,tPen\WObj:=wPaper;
    MoveL Offs(pOrigin,232.15,237.05,6.00),v60,z5,tPen\WObj:=wPaper;
    MoveL Offs(pOrigin,216.43,210.91,6.00),vTravel,z5,tPen\WObj:=wPaper;
    MoveL Offs(pOrigin,216.43,210.91,0.00),v60,z0,tPen\WObj:=wPaper;
    MoveL Offs(pOrigin,217.27,211.76,0.00),v40,z0,tPen\WObj:=wPaper;
    MoveL Offs(pOrigin,216.43,210.91,0.00),v40,fine,tPen\WObj:=wPaper;
    MoveL Offs(pOrigin,216.43,210.91,6.00),v60,z5,tPen\WObj:=wPaper;
    MoveL Offs(pOrigin,214.09,208.36,6.00),vTravel,z5,tPen\WObj:=wPaper;
    MoveL Offs(pOrigin,214.09,208.36,0.00),v60,z0,tPen\WObj:=wPaper;
    MoveL Offs(pOrigin,215.79,210.06,0.00),v40,z0,tPen\WObj:=wPaper;
    MoveL Offs(pOrigin,214.09,208.36,0.00),v40,fine,tPen\WObj:=wPaper;
    MoveL Offs(pOrigin,214.09,208.36,6.00),v60,z5,tPen\WObj:=wPaper;
    MoveL Offs(pOrigin,212.81,206.88,6.00),vTravel,z5,tPen\WObj:=wPaper;
    MoveL Offs(pOrigin,212.81,206.88,0.00),v60,z0,tPen\WObj:=wPaper;
    MoveL Offs(pOrigin,213.02,207.30,0.00),v40,z0,tPen\WObj:=wPaper;
    MoveL Offs(pOrigin,212.81,206.88,0.00),v40,fine,tPen\WObj:=wPaper;
    MoveL Offs(pOrigin,212.81,206.88,6.00),v60,z5,tPen\WObj:=wPaper;
    MoveL Offs(pOrigin,211.75,205.81,6.00),vTravel,z5,tPen\WObj:=wPaper;
    MoveL Offs(pOrigin,211.75,205.81,0.00),v60,z0,tPen\WObj:=wPaper;
    MoveL Offs(pOrigin,212.60,206.66,0.00),v40,z0,tPen\WObj:=wPaper;
    MoveL Offs(pOrigin,211.75,205.81,0.00),v40,fine,tPen\WObj:=wPaper;
    MoveL Offs(pOrigin,211.75,205.81,6.00),v60,z5,tPen\WObj:=wPaper;
    MoveL Offs(pOrigin,198.57,208.36,6.00),vTravel,z5,tPen\WObj:=wPaper;
    MoveL Offs(pOrigin,198.57,208.36,0.00),v60,z0,tPen\WObj:=wPaper;
    MoveL Offs(pOrigin,199.00,208.57,0.00),v40,z0,tPen\WObj:=wPaper;
    MoveL Offs(pOrigin,198.57,208.36,0.00),v40,fine,tPen\WObj:=wPaper;
    MoveL Offs(pOrigin,198.57,208.36,6.00),v60,z5,tPen\WObj:=wPaper;
    MoveL Offs(pOrigin,196.88,207.51,6.00),vTravel,z5,tPen\WObj:=wPaper;
    MoveL Offs(pOrigin,196.88,207.51,0.00),v60,z0,tPen\WObj:=wPaper;
    MoveL Offs(pOrigin,197.30,207.73,0.00),v40,z0,tPen\WObj:=wPaper;
    MoveL Offs(pOrigin,196.88,207.51,0.00),v40,fine,tPen\WObj:=wPaper;
    MoveL Offs(pOrigin,196.88,207.51,6.00),v60,z5,tPen\WObj:=wPaper;
    MoveL Offs(pOrigin,195.18,208.36,6.00),vTravel,z5,tPen\WObj:=wPaper;
    MoveL Offs(pOrigin,195.18,208.36,0.00),v60,z0,tPen\WObj:=wPaper;
    MoveL Offs(pOrigin,195.60,208.57,0.00),v40,z0,tPen\WObj:=wPaper;
    MoveL Offs(pOrigin,195.18,208.36,0.00),v40,fine,tPen\WObj:=wPaper;
    MoveL Offs(pOrigin,195.18,208.36,6.00),v60,z5,tPen\WObj:=wPaper;
    MoveL Offs(pOrigin,193.48,207.51,6.00),vTravel,z5,tPen\WObj:=wPaper;
    MoveL Offs(pOrigin,193.48,207.51,0.00),v60,z0,tPen\WObj:=wPaper;
    MoveL Offs(pOrigin,193.90,207.73,0.00),v40,z0,tPen\WObj:=wPaper;
    MoveL Offs(pOrigin,193.48,207.51,0.00),v40,fine,tPen\WObj:=wPaper;
    MoveL Offs(pOrigin,193.48,207.51,6.00),v60,z5,tPen\WObj:=wPaper;
    MoveL Offs(pOrigin,193.90,206.02,6.00),vTravel,z5,tPen\WObj:=wPaper;
    MoveL Offs(pOrigin,193.90,206.02,0.00),v60,z0,tPen\WObj:=wPaper;
    MoveL Offs(pOrigin,194.32,206.24,0.00),v40,z0,tPen\WObj:=wPaper;
    MoveL Offs(pOrigin,193.90,206.02,0.00),v40,z0,tPen\WObj:=wPaper;
    MoveL Offs(pOrigin,194.75,206.45,0.00),v40,z0,tPen\WObj:=wPaper;
    MoveL Offs(pOrigin,195.18,206.66,0.00),v40,z0,tPen\WObj:=wPaper;
    MoveL Offs(pOrigin,194.75,206.45,0.00),v40,fine,tPen\WObj:=wPaper;
    MoveL Offs(pOrigin,194.75,206.45,6.00),v60,z5,tPen\WObj:=wPaper;
    MoveL Offs(pOrigin,192.84,205.39,6.00),vTravel,z5,tPen\WObj:=wPaper;
    MoveL Offs(pOrigin,192.84,205.39,0.00),v60,z0,tPen\WObj:=wPaper;
    MoveL Offs(pOrigin,193.48,205.81,0.00),v40,z0,tPen\WObj:=wPaper;
    MoveL Offs(pOrigin,192.84,205.39,0.00),v40,z0,tPen\WObj:=wPaper;
    MoveL Offs(pOrigin,191.99,204.96,0.00),v40,z0,tPen\WObj:=wPaper;
    MoveL Offs(pOrigin,192.41,205.18,0.00),v40,z0,tPen\WObj:=wPaper;
    MoveL Offs(pOrigin,191.99,204.96,0.00),v40,fine,tPen\WObj:=wPaper;
    MoveL Offs(pOrigin,191.99,204.96,6.00),v60,z5,tPen\WObj:=wPaper;
    MoveL Offs(pOrigin,190.71,204.32,6.00),vTravel,z5,tPen\WObj:=wPaper;
    MoveL Offs(pOrigin,190.71,204.32,0.00),v60,z0,tPen\WObj:=wPaper;
    MoveL Offs(pOrigin,191.14,204.54,0.00),v40,z0,tPen\WObj:=wPaper;
    MoveL Offs(pOrigin,190.71,204.32,0.00),v40,fine,tPen\WObj:=wPaper;
    MoveL Offs(pOrigin,190.71,204.32,6.00),v60,z5,tPen\WObj:=wPaper;
    MoveL Offs(pOrigin,189.86,205.60,6.00),vTravel,z5,tPen\WObj:=wPaper;
    MoveL Offs(pOrigin,189.86,205.60,0.00),v60,z0,tPen\WObj:=wPaper;
    MoveL Offs(pOrigin,190.29,205.81,0.00),v40,z0,tPen\WObj:=wPaper;
    MoveL Offs(pOrigin,189.86,205.60,0.00),v40,z0,tPen\WObj:=wPaper;
    MoveL Offs(pOrigin,190.71,206.02,0.00),v40,z0,tPen\WObj:=wPaper;
    MoveL Offs(pOrigin,191.14,206.24,0.00),v40,z0,tPen\WObj:=wPaper;
    MoveL Offs(pOrigin,190.71,206.02,0.00),v40,z0,tPen\WObj:=wPaper;
    MoveL Offs(pOrigin,191.56,206.45,0.00),v40,z0,tPen\WObj:=wPaper;
    MoveL Offs(pOrigin,191.99,206.66,0.00),v40,z0,tPen\WObj:=wPaper;
    MoveL Offs(pOrigin,191.56,206.45,0.00),v40,fine,tPen\WObj:=wPaper;
    MoveL Offs(pOrigin,191.56,206.45,6.00),v60,z5,tPen\WObj:=wPaper;
    MoveL Offs(pOrigin,187.52,204.32,6.00),vTravel,z5,tPen\WObj:=wPaper;
    MoveL Offs(pOrigin,187.52,204.32,0.00),v60,z0,tPen\WObj:=wPaper;
  ENDPROC

  PROC DrawPart95()
    MoveL Offs(pOrigin,187.95,204.54,0.00),v40,z0,tPen\WObj:=wPaper;
    MoveL Offs(pOrigin,187.52,204.32,0.00),v40,fine,tPen\WObj:=wPaper;
    MoveL Offs(pOrigin,187.52,204.32,6.00),v60,z5,tPen\WObj:=wPaper;
    MoveL Offs(pOrigin,187.95,202.84,6.00),vTravel,z5,tPen\WObj:=wPaper;
    MoveL Offs(pOrigin,187.95,202.84,0.00),v60,z0,tPen\WObj:=wPaper;
    MoveL Offs(pOrigin,188.38,203.05,0.00),v40,z0,tPen\WObj:=wPaper;
    MoveL Offs(pOrigin,187.95,202.84,0.00),v40,z0,tPen\WObj:=wPaper;
    MoveL Offs(pOrigin,187.10,202.41,0.00),v40,z0,tPen\WObj:=wPaper;
    MoveL Offs(pOrigin,187.52,202.62,0.00),v40,z0,tPen\WObj:=wPaper;
    MoveL Offs(pOrigin,187.10,202.41,0.00),v40,fine,tPen\WObj:=wPaper;
    MoveL Offs(pOrigin,187.10,202.41,6.00),v60,z5,tPen\WObj:=wPaper;
    MoveL Offs(pOrigin,185.40,201.56,6.00),vTravel,z5,tPen\WObj:=wPaper;
    MoveL Offs(pOrigin,185.40,201.56,0.00),v60,z0,tPen\WObj:=wPaper;
    MoveL Offs(pOrigin,185.82,201.77,0.00),v40,z0,tPen\WObj:=wPaper;
    MoveL Offs(pOrigin,185.40,201.56,0.00),v40,fine,tPen\WObj:=wPaper;
    MoveL Offs(pOrigin,185.40,201.56,6.00),v60,z5,tPen\WObj:=wPaper;
    MoveL Offs(pOrigin,184.55,202.84,6.00),vTravel,z5,tPen\WObj:=wPaper;
    MoveL Offs(pOrigin,184.55,202.84,0.00),v60,z0,tPen\WObj:=wPaper;
    MoveL Offs(pOrigin,184.98,203.05,0.00),v40,z0,tPen\WObj:=wPaper;
    MoveL Offs(pOrigin,184.55,202.84,0.00),v40,z0,tPen\WObj:=wPaper;
    MoveL Offs(pOrigin,183.49,202.41,0.00),v40,z0,tPen\WObj:=wPaper;
    MoveL Offs(pOrigin,183.91,202.62,0.00),v40,z0,tPen\WObj:=wPaper;
    MoveL Offs(pOrigin,183.49,202.41,0.00),v40,fine,tPen\WObj:=wPaper;
    MoveL Offs(pOrigin,183.49,202.41,6.00),v60,z5,tPen\WObj:=wPaper;
    MoveL Offs(pOrigin,181.79,201.56,6.00),vTravel,z5,tPen\WObj:=wPaper;
    MoveL Offs(pOrigin,181.79,201.56,0.00),v60,z0,tPen\WObj:=wPaper;
    MoveL Offs(pOrigin,182.21,201.77,0.00),v40,z0,tPen\WObj:=wPaper;
    MoveL Offs(pOrigin,181.79,201.56,0.00),v40,fine,tPen\WObj:=wPaper;
    MoveL Offs(pOrigin,181.79,201.56,6.00),v60,z5,tPen\WObj:=wPaper;
    MoveL Offs(pOrigin,183.06,200.50,6.00),vTravel,z5,tPen\WObj:=wPaper;
    MoveL Offs(pOrigin,183.06,200.50,0.00),v60,z0,tPen\WObj:=wPaper;
    MoveL Offs(pOrigin,183.49,200.71,0.00),v40,z0,tPen\WObj:=wPaper;
    MoveL Offs(pOrigin,183.06,200.50,0.00),v40,fine,tPen\WObj:=wPaper;
    MoveL Offs(pOrigin,183.06,200.50,6.00),v60,z5,tPen\WObj:=wPaper;
    MoveL Offs(pOrigin,189.01,200.93,6.00),vTravel,z5,tPen\WObj:=wPaper;
    MoveL Offs(pOrigin,189.01,200.93,0.00),v60,z0,tPen\WObj:=wPaper;
    MoveL Offs(pOrigin,189.44,201.14,0.00),v40,z0,tPen\WObj:=wPaper;
    MoveL Offs(pOrigin,189.01,200.93,0.00),v40,fine,tPen\WObj:=wPaper;
    MoveL Offs(pOrigin,189.01,200.93,6.00),v60,z5,tPen\WObj:=wPaper;
    MoveL Offs(pOrigin,190.50,201.35,6.00),vTravel,z5,tPen\WObj:=wPaper;
    MoveL Offs(pOrigin,190.50,201.35,0.00),v60,z0,tPen\WObj:=wPaper;
    MoveL Offs(pOrigin,181.57,197.03,0.00),v40,z0,tPen\WObj:=wPaper;
    MoveL Offs(pOrigin,177.32,195.33,0.00),v40,z0,tPen\WObj:=wPaper;
    MoveL Offs(pOrigin,158.41,189.66,0.00),v40,fine,tPen\WObj:=wPaper;
    MoveL Offs(pOrigin,158.41,189.66,6.00),v60,z5,tPen\WObj:=wPaper;
    MoveL Offs(pOrigin,142.05,187.75,6.00),vTravel,z5,tPen\WObj:=wPaper;
    MoveL Offs(pOrigin,142.05,187.75,0.00),v60,z0,tPen\WObj:=wPaper;
    MoveL Offs(pOrigin,142.48,187.96,0.00),v40,z0,tPen\WObj:=wPaper;
    MoveL Offs(pOrigin,142.05,187.75,0.00),v40,fine,tPen\WObj:=wPaper;
    MoveL Offs(pOrigin,142.05,187.75,6.00),v60,z5,tPen\WObj:=wPaper;
    MoveL Offs(pOrigin,140.77,186.69,6.00),vTravel,z5,tPen\WObj:=wPaper;
    MoveL Offs(pOrigin,140.77,186.69,0.00),v60,z0,tPen\WObj:=wPaper;
    MoveL Offs(pOrigin,141.41,187.32,0.00),v40,z0,tPen\WObj:=wPaper;
    MoveL Offs(pOrigin,140.77,186.69,0.00),v40,fine,tPen\WObj:=wPaper;
    MoveL Offs(pOrigin,140.77,186.69,6.00),v60,z5,tPen\WObj:=wPaper;
    MoveL Offs(pOrigin,141.84,185.20,6.00),vTravel,z5,tPen\WObj:=wPaper;
    MoveL Offs(pOrigin,141.84,185.20,0.00),v60,z0,tPen\WObj:=wPaper;
    MoveL Offs(pOrigin,142.26,185.62,0.00),v40,z0,tPen\WObj:=wPaper;
    MoveL Offs(pOrigin,141.84,185.20,0.00),v40,fine,tPen\WObj:=wPaper;
    MoveL Offs(pOrigin,141.84,185.20,6.00),v60,z5,tPen\WObj:=wPaper;
    MoveL Offs(pOrigin,139.29,184.77,6.00),vTravel,z5,tPen\WObj:=wPaper;
    MoveL Offs(pOrigin,139.29,184.77,0.00),v60,z0,tPen\WObj:=wPaper;
    MoveL Offs(pOrigin,139.93,185.62,0.00),v40,z0,tPen\WObj:=wPaper;
    MoveL Offs(pOrigin,139.29,184.77,0.00),v40,fine,tPen\WObj:=wPaper;
    MoveL Offs(pOrigin,139.29,184.77,6.00),v60,z5,tPen\WObj:=wPaper;
    MoveL Offs(pOrigin,140.14,182.65,6.00),vTravel,z5,tPen\WObj:=wPaper;
    MoveL Offs(pOrigin,140.14,182.65,0.00),v60,z0,tPen\WObj:=wPaper;
    MoveL Offs(pOrigin,140.35,183.07,0.00),v40,z0,tPen\WObj:=wPaper;
    MoveL Offs(pOrigin,140.14,182.65,0.00),v40,fine,tPen\WObj:=wPaper;
    MoveL Offs(pOrigin,140.14,182.65,6.00),v60,z5,tPen\WObj:=wPaper;
    MoveL Offs(pOrigin,142.26,173.73,6.00),vTravel,z5,tPen\WObj:=wPaper;
    MoveL Offs(pOrigin,142.26,173.73,0.00),v60,z0,tPen\WObj:=wPaper;
    MoveL Offs(pOrigin,144.53,167.99,0.00),v40,z0,tPen\WObj:=wPaper;
    MoveL Offs(pOrigin,146.87,163.52,0.00),v40,z0,tPen\WObj:=wPaper;
    MoveL Offs(pOrigin,148.21,161.82,0.00),v40,z0,tPen\WObj:=wPaper;
    MoveL Offs(pOrigin,147.36,162.46,0.00),v40,z0,tPen\WObj:=wPaper;
    MoveL Offs(pOrigin,147.15,162.89,0.00),v40,z0,tPen\WObj:=wPaper;
    MoveL Offs(pOrigin,147.36,162.46,0.00),v40,fine,tPen\WObj:=wPaper;
    MoveL Offs(pOrigin,147.36,162.46,6.00),v60,z5,tPen\WObj:=wPaper;
    MoveL Offs(pOrigin,146.73,163.52,6.00),vTravel,z5,tPen\WObj:=wPaper;
    MoveL Offs(pOrigin,146.73,163.52,0.00),v60,z0,tPen\WObj:=wPaper;
    MoveL Offs(pOrigin,146.51,163.95,0.00),v40,z0,tPen\WObj:=wPaper;
    MoveL Offs(pOrigin,146.73,163.52,0.00),v40,z0,tPen\WObj:=wPaper;
    MoveL Offs(pOrigin,146.30,164.38,0.00),v40,z0,tPen\WObj:=wPaper;
    MoveL Offs(pOrigin,146.09,164.80,0.00),v40,z0,tPen\WObj:=wPaper;
    MoveL Offs(pOrigin,146.30,164.38,0.00),v40,z0,tPen\WObj:=wPaper;
    MoveL Offs(pOrigin,145.88,165.23,0.00),v40,z0,tPen\WObj:=wPaper;
    MoveL Offs(pOrigin,145.66,165.65,0.00),v40,z0,tPen\WObj:=wPaper;
    MoveL Offs(pOrigin,145.88,165.23,0.00),v40,fine,tPen\WObj:=wPaper;
    MoveL Offs(pOrigin,145.88,165.23,6.00),v60,z5,tPen\WObj:=wPaper;
    MoveL Offs(pOrigin,140.56,160.76,6.00),vTravel,z5,tPen\WObj:=wPaper;
    MoveL Offs(pOrigin,140.56,160.76,0.00),v60,z0,tPen\WObj:=wPaper;
    MoveL Offs(pOrigin,140.35,161.19,0.00),v40,z0,tPen\WObj:=wPaper;
    MoveL Offs(pOrigin,140.56,160.76,0.00),v40,z0,tPen\WObj:=wPaper;
    MoveL Offs(pOrigin,141.20,159.91,0.00),v40,z0,tPen\WObj:=wPaper;
    MoveL Offs(pOrigin,140.99,160.34,0.00),v40,z0,tPen\WObj:=wPaper;
    MoveL Offs(pOrigin,141.20,159.91,0.00),v40,z0,tPen\WObj:=wPaper;
    MoveL Offs(pOrigin,141.84,159.27,0.00),v40,z0,tPen\WObj:=wPaper;
    MoveL Offs(pOrigin,141.62,159.70,0.00),v40,z0,tPen\WObj:=wPaper;
    MoveL Offs(pOrigin,141.84,159.27,0.00),v40,fine,tPen\WObj:=wPaper;
    MoveL Offs(pOrigin,141.84,159.27,6.00),v60,z5,tPen\WObj:=wPaper;
    MoveL Offs(pOrigin,140.99,158.21,6.00),vTravel,z5,tPen\WObj:=wPaper;
    MoveL Offs(pOrigin,140.99,158.21,0.00),v60,z0,tPen\WObj:=wPaper;
    MoveL Offs(pOrigin,141.20,157.79,0.00),v40,z0,tPen\WObj:=wPaper;
    MoveL Offs(pOrigin,140.99,158.21,0.00),v40,z0,tPen\WObj:=wPaper;
    MoveL Offs(pOrigin,141.62,157.57,0.00),v40,z0,tPen\WObj:=wPaper;
    MoveL Offs(pOrigin,141.84,157.15,0.00),v40,z0,tPen\WObj:=wPaper;
    MoveL Offs(pOrigin,141.62,157.57,0.00),v40,z0,tPen\WObj:=wPaper;
    MoveL Offs(pOrigin,142.26,156.94,0.00),v40,z0,tPen\WObj:=wPaper;
    MoveL Offs(pOrigin,142.48,156.51,0.00),v40,z0,tPen\WObj:=wPaper;
    MoveL Offs(pOrigin,142.26,156.94,0.00),v40,fine,tPen\WObj:=wPaper;
    MoveL Offs(pOrigin,142.26,156.94,6.00),v60,z5,tPen\WObj:=wPaper;
    MoveL Offs(pOrigin,143.32,157.57,6.00),vTravel,z5,tPen\WObj:=wPaper;
    MoveL Offs(pOrigin,143.32,157.57,0.00),v60,z0,tPen\WObj:=wPaper;
    MoveL Offs(pOrigin,143.11,158.00,0.00),v40,z0,tPen\WObj:=wPaper;
    MoveL Offs(pOrigin,143.32,157.57,0.00),v40,z0,tPen\WObj:=wPaper;
    MoveL Offs(pOrigin,143.96,156.94,0.00),v40,z0,tPen\WObj:=wPaper;
    MoveL Offs(pOrigin,143.75,157.36,0.00),v40,z0,tPen\WObj:=wPaper;
    MoveL Offs(pOrigin,143.96,156.94,0.00),v40,fine,tPen\WObj:=wPaper;
    MoveL Offs(pOrigin,143.96,156.94,6.00),v60,z5,tPen\WObj:=wPaper;
  ENDPROC

  PROC DrawPart96()
    MoveL Offs(pOrigin,143.11,155.88,6.00),vTravel,z5,tPen\WObj:=wPaper;
    MoveL Offs(pOrigin,143.11,155.88,0.00),v60,z0,tPen\WObj:=wPaper;
    MoveL Offs(pOrigin,142.90,156.30,0.00),v40,z0,tPen\WObj:=wPaper;
    MoveL Offs(pOrigin,143.11,155.88,0.00),v40,z0,tPen\WObj:=wPaper;
    MoveL Offs(pOrigin,143.75,155.24,0.00),v40,z0,tPen\WObj:=wPaper;
    MoveL Offs(pOrigin,143.54,155.66,0.00),v40,z0,tPen\WObj:=wPaper;
    MoveL Offs(pOrigin,143.75,155.24,0.00),v40,z0,tPen\WObj:=wPaper;
    MoveL Offs(pOrigin,144.18,155.02,0.00),v40,z0,tPen\WObj:=wPaper;
    MoveL Offs(pOrigin,144.39,154.60,0.00),v40,z0,tPen\WObj:=wPaper;
    MoveL Offs(pOrigin,144.18,155.02,0.00),v40,z0,tPen\WObj:=wPaper;
    MoveL Offs(pOrigin,144.81,154.39,0.00),v40,z0,tPen\WObj:=wPaper;
    MoveL Offs(pOrigin,145.24,153.96,0.00),v40,z0,tPen\WObj:=wPaper;
    MoveL Offs(pOrigin,144.81,154.39,0.00),v40,z0,tPen\WObj:=wPaper;
    MoveL Offs(pOrigin,145.66,153.75,0.00),v40,z0,tPen\WObj:=wPaper;
    MoveL Offs(pOrigin,145.88,153.32,0.00),v40,z0,tPen\WObj:=wPaper;
    MoveL Offs(pOrigin,145.66,153.75,0.00),v40,z0,tPen\WObj:=wPaper;
    MoveL Offs(pOrigin,146.30,154.39,0.00),v40,z0,tPen\WObj:=wPaper;
    MoveL Offs(pOrigin,146.09,154.81,0.00),v40,z0,tPen\WObj:=wPaper;
    MoveL Offs(pOrigin,146.30,154.39,0.00),v40,z0,tPen\WObj:=wPaper;
    MoveL Offs(pOrigin,146.73,154.18,0.00),v40,z0,tPen\WObj:=wPaper;
    MoveL Offs(pOrigin,146.94,153.75,0.00),v40,z0,tPen\WObj:=wPaper;
    MoveL Offs(pOrigin,146.73,154.18,0.00),v40,fine,tPen\WObj:=wPaper;
    MoveL Offs(pOrigin,146.73,154.18,6.00),v60,z5,tPen\WObj:=wPaper;
    MoveL Offs(pOrigin,145.66,155.02,6.00),vTravel,z5,tPen\WObj:=wPaper;
    MoveL Offs(pOrigin,145.66,155.02,0.00),v60,z0,tPen\WObj:=wPaper;
    MoveL Offs(pOrigin,145.45,155.45,0.00),v40,z0,tPen\WObj:=wPaper;
    MoveL Offs(pOrigin,145.66,155.02,0.00),v40,z0,tPen\WObj:=wPaper;
    MoveL Offs(pOrigin,145.02,155.66,0.00),v40,z0,tPen\WObj:=wPaper;
    MoveL Offs(pOrigin,144.81,156.09,0.00),v40,z0,tPen\WObj:=wPaper;
    MoveL Offs(pOrigin,145.02,155.66,0.00),v40,fine,tPen\WObj:=wPaper;
    MoveL Offs(pOrigin,145.02,155.66,6.00),v60,z5,tPen\WObj:=wPaper;
    MoveL Offs(pOrigin,142.69,158.21,6.00),vTravel,z5,tPen\WObj:=wPaper;
    MoveL Offs(pOrigin,142.69,158.21,0.00),v60,z0,tPen\WObj:=wPaper;
    MoveL Offs(pOrigin,142.48,158.64,0.00),v40,z0,tPen\WObj:=wPaper;
    MoveL Offs(pOrigin,142.69,158.21,0.00),v40,fine,tPen\WObj:=wPaper;
    MoveL Offs(pOrigin,142.69,158.21,6.00),v60,z5,tPen\WObj:=wPaper;
    MoveL Offs(pOrigin,139.93,159.49,6.00),vTravel,z5,tPen\WObj:=wPaper;
    MoveL Offs(pOrigin,139.93,159.49,0.00),v60,z0,tPen\WObj:=wPaper;
    MoveL Offs(pOrigin,140.14,159.06,0.00),v40,z0,tPen\WObj:=wPaper;
    MoveL Offs(pOrigin,139.93,159.49,0.00),v40,z0,tPen\WObj:=wPaper;
    MoveL Offs(pOrigin,139.50,159.70,0.00),v40,z0,tPen\WObj:=wPaper;
    MoveL Offs(pOrigin,139.29,160.12,0.00),v40,z0,tPen\WObj:=wPaper;
    MoveL Offs(pOrigin,139.50,159.70,0.00),v40,fine,tPen\WObj:=wPaper;
    MoveL Offs(pOrigin,139.50,159.70,6.00),v60,z5,tPen\WObj:=wPaper;
    MoveL Offs(pOrigin,138.65,160.98,6.00),vTravel,z5,tPen\WObj:=wPaper;
    MoveL Offs(pOrigin,138.65,160.98,0.00),v60,z0,tPen\WObj:=wPaper;
    MoveL Offs(pOrigin,138.86,160.55,0.00),v40,z0,tPen\WObj:=wPaper;
    MoveL Offs(pOrigin,138.65,160.98,0.00),v40,z0,tPen\WObj:=wPaper;
    MoveL Offs(pOrigin,138.01,161.82,0.00),v40,z0,tPen\WObj:=wPaper;
    MoveL Offs(pOrigin,138.23,161.40,0.00),v40,z0,tPen\WObj:=wPaper;
    MoveL Offs(pOrigin,138.01,161.82,0.00),v40,fine,tPen\WObj:=wPaper;
    MoveL Offs(pOrigin,138.01,161.82,6.00),v60,z5,tPen\WObj:=wPaper;
    MoveL Offs(pOrigin,139.93,161.61,6.00),vTravel,z5,tPen\WObj:=wPaper;
    MoveL Offs(pOrigin,139.93,161.61,0.00),v60,z0,tPen\WObj:=wPaper;
    MoveL Offs(pOrigin,139.71,162.04,0.00),v40,z0,tPen\WObj:=wPaper;
    MoveL Offs(pOrigin,139.93,161.61,0.00),v40,fine,tPen\WObj:=wPaper;
    MoveL Offs(pOrigin,139.93,161.61,6.00),v60,z5,tPen\WObj:=wPaper;
    MoveL Offs(pOrigin,137.80,164.59,6.00),vTravel,z5,tPen\WObj:=wPaper;
    MoveL Offs(pOrigin,137.80,164.59,0.00),v60,z0,tPen\WObj:=wPaper;
    MoveL Offs(pOrigin,137.59,165.01,0.00),v40,z0,tPen\WObj:=wPaper;
    MoveL Offs(pOrigin,137.80,164.59,0.00),v40,fine,tPen\WObj:=wPaper;
    MoveL Offs(pOrigin,137.80,164.59,6.00),v60,z5,tPen\WObj:=wPaper;
    MoveL Offs(pOrigin,137.16,165.65,6.00),vTravel,z5,tPen\WObj:=wPaper;
    MoveL Offs(pOrigin,137.16,165.65,0.00),v60,z0,tPen\WObj:=wPaper;
    MoveL Offs(pOrigin,136.95,166.07,0.00),v40,z0,tPen\WObj:=wPaper;
    MoveL Offs(pOrigin,137.16,165.65,0.00),v40,fine,tPen\WObj:=wPaper;
    MoveL Offs(pOrigin,137.16,165.65,6.00),v60,z5,tPen\WObj:=wPaper;
    MoveL Offs(pOrigin,136.10,164.59,6.00),vTravel,z5,tPen\WObj:=wPaper;
    MoveL Offs(pOrigin,136.10,164.59,0.00),v60,z0,tPen\WObj:=wPaper;
    MoveL Offs(pOrigin,135.89,165.01,0.00),v40,z0,tPen\WObj:=wPaper;
    MoveL Offs(pOrigin,136.10,164.59,0.00),v40,fine,tPen\WObj:=wPaper;
    MoveL Offs(pOrigin,136.10,164.59,6.00),v60,z5,tPen\WObj:=wPaper;
    MoveL Offs(pOrigin,149.91,157.15,6.00),vTravel,z5,tPen\WObj:=wPaper;
    MoveL Offs(pOrigin,149.91,157.15,0.00),v60,z0,tPen\WObj:=wPaper;
    MoveL Offs(pOrigin,149.70,157.57,0.00),v40,z0,tPen\WObj:=wPaper;
    MoveL Offs(pOrigin,149.91,157.15,0.00),v40,fine,tPen\WObj:=wPaper;
    MoveL Offs(pOrigin,149.91,157.15,6.00),v60,z5,tPen\WObj:=wPaper;
    MoveL Offs(pOrigin,150.55,156.09,6.00),vTravel,z5,tPen\WObj:=wPaper;
    MoveL Offs(pOrigin,150.55,156.09,0.00),v60,z0,tPen\WObj:=wPaper;
    MoveL Offs(pOrigin,150.34,156.51,0.00),v40,z0,tPen\WObj:=wPaper;
    MoveL Offs(pOrigin,150.55,156.09,0.00),v40,fine,tPen\WObj:=wPaper;
    MoveL Offs(pOrigin,150.55,156.09,6.00),v60,z5,tPen\WObj:=wPaper;
    MoveL Offs(pOrigin,148.00,152.26,6.00),vTravel,z5,tPen\WObj:=wPaper;
    MoveL Offs(pOrigin,148.00,152.26,0.00),v60,z0,tPen\WObj:=wPaper;
    MoveL Offs(pOrigin,149.91,150.35,0.00),v40,fine,tPen\WObj:=wPaper;
    MoveL Offs(pOrigin,149.91,150.35,6.00),v60,z5,tPen\WObj:=wPaper;
    MoveL Offs(pOrigin,151.40,138.45,6.00),vTravel,z5,tPen\WObj:=wPaper;
    MoveL Offs(pOrigin,151.40,138.45,0.00),v60,z0,tPen\WObj:=wPaper;
    MoveL Offs(pOrigin,151.19,138.66,0.00),v40,z0,tPen\WObj:=wPaper;
    MoveL Offs(pOrigin,151.40,138.24,0.00),v40,z0,tPen\WObj:=wPaper;
    MoveL Offs(pOrigin,152.68,137.81,0.00),v40,z0,tPen\WObj:=wPaper;
    MoveL Offs(pOrigin,152.68,138.02,0.00),v40,z0,tPen\WObj:=wPaper;
    MoveL Offs(pOrigin,152.68,138.02,0.00),v40,z0,tPen\WObj:=wPaper;
    MoveL Offs(pOrigin,154.59,136.11,0.00),v40,z0,tPen\WObj:=wPaper;
    MoveL Offs(pOrigin,155.01,135.05,0.00),v40,z0,tPen\WObj:=wPaper;
    MoveL Offs(pOrigin,157.85,131.86,0.00),v40,z0,tPen\WObj:=wPaper;
    MoveL Offs(pOrigin,158.20,129.95,0.00),v40,z0,tPen\WObj:=wPaper;
    MoveL Offs(pOrigin,157.35,130.16,0.00),v40,fine,tPen\WObj:=wPaper;
    MoveL Offs(pOrigin,157.35,130.16,6.00),v60,z5,tPen\WObj:=wPaper;
    MoveL Offs(pOrigin,156.29,130.80,6.00),vTravel,z5,tPen\WObj:=wPaper;
    MoveL Offs(pOrigin,156.29,130.80,0.00),v60,z0,tPen\WObj:=wPaper;
    MoveL Offs(pOrigin,156.78,130.45,0.00),v40,z0,tPen\WObj:=wPaper;
    MoveL Offs(pOrigin,151.40,134.06,0.00),v40,z0,tPen\WObj:=wPaper;
    MoveL Offs(pOrigin,148.00,135.55,0.00),v40,z0,tPen\WObj:=wPaper;
    MoveL Offs(pOrigin,143.75,136.75,0.00),v40,fine,tPen\WObj:=wPaper;
    MoveL Offs(pOrigin,143.75,136.75,6.00),v60,z5,tPen\WObj:=wPaper;
    MoveL Offs(pOrigin,154.16,136.32,6.00),vTravel,z5,tPen\WObj:=wPaper;
    MoveL Offs(pOrigin,154.16,136.32,0.00),v60,z0,tPen\WObj:=wPaper;
    MoveL Offs(pOrigin,153.74,136.75,0.00),v40,z0,tPen\WObj:=wPaper;
    MoveL Offs(pOrigin,154.16,136.32,0.00),v40,fine,tPen\WObj:=wPaper;
    MoveL Offs(pOrigin,154.16,136.32,6.00),v60,z5,tPen\WObj:=wPaper;
    MoveL Offs(pOrigin,156.93,132.93,6.00),vTravel,z5,tPen\WObj:=wPaper;
    MoveL Offs(pOrigin,156.93,132.93,0.00),v60,z0,tPen\WObj:=wPaper;
    MoveL Offs(pOrigin,155.01,134.84,0.00),v40,z0,tPen\WObj:=wPaper;
    MoveL Offs(pOrigin,156.93,132.93,0.00),v40,fine,tPen\WObj:=wPaper;
    MoveL Offs(pOrigin,156.93,132.93,6.00),v60,z5,tPen\WObj:=wPaper;
    MoveL Offs(pOrigin,131.64,124.21,6.00),vTravel,z5,tPen\WObj:=wPaper;
    MoveL Offs(pOrigin,131.64,124.21,0.00),v60,z0,tPen\WObj:=wPaper;
    MoveL Offs(pOrigin,131.43,123.57,0.00),v40,z0,tPen\WObj:=wPaper;
    MoveL Offs(pOrigin,129.30,121.66,0.00),v40,z0,tPen\WObj:=wPaper;
  ENDPROC

  PROC DrawPart97()
    MoveL Offs(pOrigin,116.97,114.44,0.00),v40,fine,tPen\WObj:=wPaper;
    MoveL Offs(pOrigin,116.97,114.44,6.00),v60,z5,tPen\WObj:=wPaper;
    MoveL Offs(pOrigin,119.10,112.10,6.00),vTravel,z5,tPen\WObj:=wPaper;
    MoveL Offs(pOrigin,119.10,112.10,0.00),v60,z0,tPen\WObj:=wPaper;
    MoveL Offs(pOrigin,118.04,112.10,0.00),v40,z0,tPen\WObj:=wPaper;
    MoveL Offs(pOrigin,117.82,111.46,0.00),v40,z0,tPen\WObj:=wPaper;
    MoveL Offs(pOrigin,117.40,111.25,0.00),v40,z0,tPen\WObj:=wPaper;
    MoveL Offs(pOrigin,117.40,111.25,0.00),v40,z0,tPen\WObj:=wPaper;
    MoveL Offs(pOrigin,117.19,110.40,0.00),v40,z0,tPen\WObj:=wPaper;
    MoveL Offs(pOrigin,116.12,110.40,0.00),v40,z0,tPen\WObj:=wPaper;
    MoveL Offs(pOrigin,116.12,110.40,0.00),v40,z0,tPen\WObj:=wPaper;
    MoveL Offs(pOrigin,116.55,111.25,0.00),v40,z0,tPen\WObj:=wPaper;
    MoveL Offs(pOrigin,117.19,111.46,0.00),v40,z0,tPen\WObj:=wPaper;
    MoveL Offs(pOrigin,117.40,111.25,0.00),v40,z0,tPen\WObj:=wPaper;
    MoveL Offs(pOrigin,117.82,111.25,0.00),v40,z0,tPen\WObj:=wPaper;
    MoveL Offs(pOrigin,118.68,111.32,0.00),v40,z0,tPen\WObj:=wPaper;
    MoveL Offs(pOrigin,119.31,112.10,0.00),v40,z0,tPen\WObj:=wPaper;
    MoveL Offs(pOrigin,120.38,112.60,0.00),v40,z0,tPen\WObj:=wPaper;
    MoveL Offs(pOrigin,127.81,114.65,0.00),v40,fine,tPen\WObj:=wPaper;
    MoveL Offs(pOrigin,127.81,114.65,6.00),v60,z5,tPen\WObj:=wPaper;
    MoveL Offs(pOrigin,116.12,110.40,6.00),vTravel,z5,tPen\WObj:=wPaper;
    MoveL Offs(pOrigin,116.12,110.40,0.00),v60,z0,tPen\WObj:=wPaper;
    MoveL Offs(pOrigin,114.64,109.55,0.00),v40,fine,tPen\WObj:=wPaper;
    MoveL Offs(pOrigin,114.64,109.55,6.00),v60,z5,tPen\WObj:=wPaper;
    MoveL Offs(pOrigin,127.18,90.00,6.00),vTravel,z5,tPen\WObj:=wPaper;
    MoveL Offs(pOrigin,127.18,90.00,0.00),v60,z0,tPen\WObj:=wPaper;
    MoveL Offs(pOrigin,128.88,90.07,0.00),v40,z0,tPen\WObj:=wPaper;
    MoveL Offs(pOrigin,133.12,88.87,0.00),v40,z0,tPen\WObj:=wPaper;
    MoveL Offs(pOrigin,133.98,88.30,0.00),v40,z0,tPen\WObj:=wPaper;
    MoveL Offs(pOrigin,134.61,87.31,0.00),v40,z0,tPen\WObj:=wPaper;
    MoveL Offs(pOrigin,136.10,86.88,0.00),v40,z0,tPen\WObj:=wPaper;
    MoveL Offs(pOrigin,139.07,85.32,0.00),v40,z0,tPen\WObj:=wPaper;
    MoveL Offs(pOrigin,139.07,85.32,0.00),v40,z0,tPen\WObj:=wPaper;
    MoveL Offs(pOrigin,139.50,84.47,0.00),v40,z0,tPen\WObj:=wPaper;
    MoveL Offs(pOrigin,140.77,83.84,0.00),v40,z0,tPen\WObj:=wPaper;
    MoveL Offs(pOrigin,140.99,83.41,0.00),v40,z0,tPen\WObj:=wPaper;
    MoveL Offs(pOrigin,140.99,83.41,0.00),v40,z0,tPen\WObj:=wPaper;
    MoveL Offs(pOrigin,140.35,83.20,0.00),v40,z0,tPen\WObj:=wPaper;
    MoveL Offs(pOrigin,132.91,84.26,0.00),v40,z0,tPen\WObj:=wPaper;
    MoveL Offs(pOrigin,126.96,84.05,0.00),v40,z0,tPen\WObj:=wPaper;
    MoveL Offs(pOrigin,121.65,82.99,0.00),v40,z0,tPen\WObj:=wPaper;
    MoveL Offs(pOrigin,117.40,81.29,0.00),v40,z0,tPen\WObj:=wPaper;
    MoveL Offs(pOrigin,117.26,80.86,0.00),v40,z0,tPen\WObj:=wPaper;
    MoveL Offs(pOrigin,117.82,80.65,0.00),v40,z0,tPen\WObj:=wPaper;
    MoveL Offs(pOrigin,123.78,82.56,0.00),v40,z0,tPen\WObj:=wPaper;
    MoveL Offs(pOrigin,125.26,82.78,0.00),v40,z0,tPen\WObj:=wPaper;
    MoveL Offs(pOrigin,125.90,82.35,0.00),v40,fine,tPen\WObj:=wPaper;
    MoveL Offs(pOrigin,125.90,82.35,6.00),v60,z5,tPen\WObj:=wPaper;
    MoveL Offs(pOrigin,120.59,79.38,6.00),vTravel,z5,tPen\WObj:=wPaper;
    MoveL Offs(pOrigin,120.59,79.38,0.00),v60,z0,tPen\WObj:=wPaper;
    MoveL Offs(pOrigin,121.01,79.59,0.00),v40,z0,tPen\WObj:=wPaper;
    MoveL Offs(pOrigin,120.59,79.38,0.00),v40,fine,tPen\WObj:=wPaper;
    MoveL Offs(pOrigin,120.59,79.38,6.00),v60,z5,tPen\WObj:=wPaper;
    MoveL Offs(pOrigin,117.19,80.65,6.00),vTravel,z5,tPen\WObj:=wPaper;
    MoveL Offs(pOrigin,117.19,80.65,0.00),v60,z0,tPen\WObj:=wPaper;
    MoveL Offs(pOrigin,116.12,80.30,0.00),v40,z0,tPen\WObj:=wPaper;
    MoveL Offs(pOrigin,112.30,77.46,0.00),v40,z0,tPen\WObj:=wPaper;
    MoveL Offs(pOrigin,106.99,70.88,0.00),v40,z0,tPen\WObj:=wPaper;
    MoveL Offs(pOrigin,101.89,65.99,0.00),v40,z0,tPen\WObj:=wPaper;
    MoveL Offs(pOrigin,100.40,65.56,0.00),v40,z0,tPen\WObj:=wPaper;
    MoveL Offs(pOrigin,100.40,65.56,0.00),v40,z0,tPen\WObj:=wPaper;
    MoveL Offs(pOrigin,100.12,64.07,0.00),v40,z0,tPen\WObj:=wPaper;
    MoveL Offs(pOrigin,99.20,63.44,0.00),v40,z0,tPen\WObj:=wPaper;
    MoveL Offs(pOrigin,97.35,59.83,0.00),v40,z0,tPen\WObj:=wPaper;
    MoveL Offs(pOrigin,97.35,58.76,0.00),v40,z0,tPen\WObj:=wPaper;
    MoveL Offs(pOrigin,96.43,57.91,0.00),v40,z0,tPen\WObj:=wPaper;
    MoveL Offs(pOrigin,95.94,56.21,0.00),v40,z0,tPen\WObj:=wPaper;
    MoveL Offs(pOrigin,95.94,56.21,0.00),v40,z0,tPen\WObj:=wPaper;
    MoveL Offs(pOrigin,95.87,55.36,0.00),v40,z0,tPen\WObj:=wPaper;
    MoveL Offs(pOrigin,94.73,54.51,0.00),v40,z0,tPen\WObj:=wPaper;
    MoveL Offs(pOrigin,94.45,52.81,0.00),v40,z0,tPen\WObj:=wPaper;
    MoveL Offs(pOrigin,94.45,52.81,0.00),v40,z0,tPen\WObj:=wPaper;
    MoveL Offs(pOrigin,94.66,51.96,0.00),v40,z0,tPen\WObj:=wPaper;
    MoveL Offs(pOrigin,94.24,50.05,0.00),v40,z0,tPen\WObj:=wPaper;
    MoveL Offs(pOrigin,94.24,48.14,0.00),v40,z0,tPen\WObj:=wPaper;
    MoveL Offs(pOrigin,94.59,46.86,0.00),v40,z0,tPen\WObj:=wPaper;
    MoveL Offs(pOrigin,95.72,45.16,0.00),v40,z0,tPen\WObj:=wPaper;
    MoveL Offs(pOrigin,98.28,42.83,0.00),v40,z0,tPen\WObj:=wPaper;
    MoveL Offs(pOrigin,98.91,42.61,0.00),v40,z0,tPen\WObj:=wPaper;
    MoveL Offs(pOrigin,99.97,41.90,0.00),v40,z0,tPen\WObj:=wPaper;
    MoveL Offs(pOrigin,102.74,40.91,0.00),v40,z0,tPen\WObj:=wPaper;
    MoveL Offs(pOrigin,105.50,40.28,0.00),v40,z0,tPen\WObj:=wPaper;
    MoveL Offs(pOrigin,106.70,40.35,0.00),v40,z0,tPen\WObj:=wPaper;
    MoveL Offs(pOrigin,106.63,41.34,0.00),v40,z0,tPen\WObj:=wPaper;
    MoveL Offs(pOrigin,105.43,43.46,0.00),v40,z0,tPen\WObj:=wPaper;
    MoveL Offs(pOrigin,104.86,45.59,0.00),v40,z0,tPen\WObj:=wPaper;
    MoveL Offs(pOrigin,104.86,49.84,0.00),v40,z0,tPen\WObj:=wPaper;
    MoveL Offs(pOrigin,105.29,50.47,0.00),v40,fine,tPen\WObj:=wPaper;
    MoveL Offs(pOrigin,105.29,50.47,6.00),v60,z5,tPen\WObj:=wPaper;
    MoveL Offs(pOrigin,99.34,42.40,6.00),vTravel,z5,tPen\WObj:=wPaper;
    MoveL Offs(pOrigin,99.34,42.40,0.00),v60,z0,tPen\WObj:=wPaper;
    MoveL Offs(pOrigin,99.76,42.19,0.00),v40,z0,tPen\WObj:=wPaper;
    MoveL Offs(pOrigin,99.34,42.40,0.00),v40,fine,tPen\WObj:=wPaper;
    MoveL Offs(pOrigin,99.34,42.40,6.00),v60,z5,tPen\WObj:=wPaper;
    MoveL Offs(pOrigin,99.34,40.70,6.00),vTravel,z5,tPen\WObj:=wPaper;
    MoveL Offs(pOrigin,99.34,40.70,0.00),v60,z0,tPen\WObj:=wPaper;
    MoveL Offs(pOrigin,99.76,40.49,0.00),v40,z0,tPen\WObj:=wPaper;
    MoveL Offs(pOrigin,99.34,40.70,0.00),v40,fine,tPen\WObj:=wPaper;
    MoveL Offs(pOrigin,99.34,40.70,6.00),v60,z5,tPen\WObj:=wPaper;
    MoveL Offs(pOrigin,97.00,43.67,6.00),vTravel,z5,tPen\WObj:=wPaper;
    MoveL Offs(pOrigin,97.00,43.67,0.00),v60,z0,tPen\WObj:=wPaper;
    MoveL Offs(pOrigin,95.51,45.16,0.00),v40,z0,tPen\WObj:=wPaper;
    MoveL Offs(pOrigin,97.00,43.67,0.00),v40,fine,tPen\WObj:=wPaper;
    MoveL Offs(pOrigin,97.00,43.67,6.00),v60,z5,tPen\WObj:=wPaper;
    MoveL Offs(pOrigin,95.94,42.61,6.00),vTravel,z5,tPen\WObj:=wPaper;
    MoveL Offs(pOrigin,95.94,42.61,0.00),v60,z0,tPen\WObj:=wPaper;
    MoveL Offs(pOrigin,94.03,44.53,0.00),v40,z0,tPen\WObj:=wPaper;
    MoveL Offs(pOrigin,95.94,42.61,0.00),v40,fine,tPen\WObj:=wPaper;
    MoveL Offs(pOrigin,95.94,42.61,6.00),v60,z5,tPen\WObj:=wPaper;
    MoveL Offs(pOrigin,93.60,45.16,6.00),vTravel,z5,tPen\WObj:=wPaper;
    MoveL Offs(pOrigin,93.60,45.16,0.00),v60,z0,tPen\WObj:=wPaper;
    MoveL Offs(pOrigin,93.39,45.59,0.00),v40,z0,tPen\WObj:=wPaper;
    MoveL Offs(pOrigin,93.60,45.16,0.00),v40,fine,tPen\WObj:=wPaper;
    MoveL Offs(pOrigin,93.60,45.16,6.00),v60,z5,tPen\WObj:=wPaper;
    MoveL Offs(pOrigin,94.66,54.72,6.00),vTravel,z5,tPen\WObj:=wPaper;
    MoveL Offs(pOrigin,94.66,54.72,0.00),v60,z0,tPen\WObj:=wPaper;
    MoveL Offs(pOrigin,94.66,55.36,0.00),v40,z0,tPen\WObj:=wPaper;
    MoveL Offs(pOrigin,95.51,56.21,0.00),v40,z0,tPen\WObj:=wPaper;
    MoveL Offs(pOrigin,95.94,56.21,0.00),v40,fine,tPen\WObj:=wPaper;
    MoveL Offs(pOrigin,95.94,56.21,6.00),v60,z5,tPen\WObj:=wPaper;
  ENDPROC

  PROC DrawPart98()
    MoveL Offs(pOrigin,94.66,55.58,6.00),vTravel,z5,tPen\WObj:=wPaper;
    MoveL Offs(pOrigin,94.66,55.58,0.00),v60,z0,tPen\WObj:=wPaper;
    MoveL Offs(pOrigin,94.45,56.21,0.00),v40,z0,tPen\WObj:=wPaper;
    MoveL Offs(pOrigin,96.36,61.53,0.00),v40,z0,tPen\WObj:=wPaper;
    MoveL Offs(pOrigin,96.36,62.38,0.00),v40,fine,tPen\WObj:=wPaper;
    MoveL Offs(pOrigin,96.36,62.38,6.00),v60,z5,tPen\WObj:=wPaper;
    MoveL Offs(pOrigin,94.88,60.89,6.00),vTravel,z5,tPen\WObj:=wPaper;
    MoveL Offs(pOrigin,94.88,60.89,0.00),v60,z0,tPen\WObj:=wPaper;
    MoveL Offs(pOrigin,95.09,61.31,0.00),v40,z0,tPen\WObj:=wPaper;
    MoveL Offs(pOrigin,94.88,60.89,0.00),v40,z0,tPen\WObj:=wPaper;
    MoveL Offs(pOrigin,94.45,60.04,0.00),v40,z0,tPen\WObj:=wPaper;
    MoveL Offs(pOrigin,94.66,60.46,0.00),v40,z0,tPen\WObj:=wPaper;
    MoveL Offs(pOrigin,94.45,60.04,0.00),v40,fine,tPen\WObj:=wPaper;
    MoveL Offs(pOrigin,94.45,60.04,6.00),v60,z5,tPen\WObj:=wPaper;
    MoveL Offs(pOrigin,96.57,58.34,6.00),vTravel,z5,tPen\WObj:=wPaper;
    MoveL Offs(pOrigin,96.57,58.34,0.00),v60,z0,tPen\WObj:=wPaper;
    MoveL Offs(pOrigin,96.79,59.61,0.00),v40,z0,tPen\WObj:=wPaper;
    MoveL Offs(pOrigin,97.21,59.61,0.00),v40,fine,tPen\WObj:=wPaper;
    MoveL Offs(pOrigin,97.21,59.61,6.00),v60,z5,tPen\WObj:=wPaper;
    MoveL Offs(pOrigin,85.53,32.62,6.00),vTravel,z5,tPen\WObj:=wPaper;
    MoveL Offs(pOrigin,85.53,32.62,0.00),v60,z0,tPen\WObj:=wPaper;
    MoveL Offs(pOrigin,85.95,33.05,0.00),v40,z0,tPen\WObj:=wPaper;
    MoveL Offs(pOrigin,85.53,32.62,0.00),v40,fine,tPen\WObj:=wPaper;
    MoveL Offs(pOrigin,85.53,32.62,6.00),v60,z5,tPen\WObj:=wPaper;
    MoveL Offs(pOrigin,116.34,36.24,6.00),vTravel,z5,tPen\WObj:=wPaper;
    MoveL Offs(pOrigin,116.34,36.24,0.00),v60,z0,tPen\WObj:=wPaper;
    MoveL Offs(pOrigin,116.55,35.81,0.00),v40,z0,tPen\WObj:=wPaper;
    MoveL Offs(pOrigin,117.19,35.81,0.00),v40,z0,tPen\WObj:=wPaper;
    MoveL Offs(pOrigin,117.61,36.45,0.00),v40,fine,tPen\WObj:=wPaper;
    MoveL Offs(pOrigin,117.61,36.45,6.00),v60,z5,tPen\WObj:=wPaper;
    MoveL Offs(pOrigin,122.29,40.49,6.00),vTravel,z5,tPen\WObj:=wPaper;
    MoveL Offs(pOrigin,122.29,40.49,0.00),v60,z0,tPen\WObj:=wPaper;
    MoveL Offs(pOrigin,121.65,41.97,0.00),v40,fine,tPen\WObj:=wPaper;
    MoveL Offs(pOrigin,121.65,41.97,6.00),v60,z5,tPen\WObj:=wPaper;
    MoveL Offs(pOrigin,122.50,43.04,6.00),vTravel,z5,tPen\WObj:=wPaper;
    MoveL Offs(pOrigin,122.50,43.04,0.00),v60,z0,tPen\WObj:=wPaper;
    MoveL Offs(pOrigin,122.29,43.46,0.00),v40,z0,tPen\WObj:=wPaper;
    MoveL Offs(pOrigin,122.50,43.04,0.00),v40,z0,tPen\WObj:=wPaper;
    MoveL Offs(pOrigin,122.07,43.89,0.00),v40,z0,tPen\WObj:=wPaper;
    MoveL Offs(pOrigin,121.86,44.31,0.00),v40,z0,tPen\WObj:=wPaper;
    MoveL Offs(pOrigin,122.07,43.89,0.00),v40,fine,tPen\WObj:=wPaper;
    MoveL Offs(pOrigin,122.07,43.89,6.00),v60,z5,tPen\WObj:=wPaper;
    MoveL Offs(pOrigin,123.14,42.19,6.00),vTravel,z5,tPen\WObj:=wPaper;
    MoveL Offs(pOrigin,123.14,42.19,0.00),v60,z0,tPen\WObj:=wPaper;
    MoveL Offs(pOrigin,122.71,42.61,0.00),v40,z0,tPen\WObj:=wPaper;
    MoveL Offs(pOrigin,123.14,42.19,0.00),v40,fine,tPen\WObj:=wPaper;
    MoveL Offs(pOrigin,123.14,42.19,6.00),v60,z5,tPen\WObj:=wPaper;
    MoveL Offs(pOrigin,125.26,42.19,6.00),vTravel,z5,tPen\WObj:=wPaper;
    MoveL Offs(pOrigin,125.26,42.19,0.00),v60,z0,tPen\WObj:=wPaper;
    MoveL Offs(pOrigin,125.05,42.61,0.00),v40,z0,tPen\WObj:=wPaper;
    MoveL Offs(pOrigin,125.26,42.19,0.00),v40,z0,tPen\WObj:=wPaper;
    MoveL Offs(pOrigin,125.90,41.55,0.00),v40,z0,tPen\WObj:=wPaper;
    MoveL Offs(pOrigin,126.11,41.12,0.00),v40,z0,tPen\WObj:=wPaper;
    MoveL Offs(pOrigin,125.90,41.55,0.00),v40,fine,tPen\WObj:=wPaper;
    MoveL Offs(pOrigin,125.90,41.55,6.00),v60,z5,tPen\WObj:=wPaper;
    MoveL Offs(pOrigin,124.62,40.49,6.00),vTravel,z5,tPen\WObj:=wPaper;
    MoveL Offs(pOrigin,124.62,40.49,0.00),v60,z0,tPen\WObj:=wPaper;
    MoveL Offs(pOrigin,123.35,41.76,0.00),v40,z0,tPen\WObj:=wPaper;
    MoveL Offs(pOrigin,124.62,40.49,0.00),v40,fine,tPen\WObj:=wPaper;
    MoveL Offs(pOrigin,124.62,40.49,6.00),v60,z5,tPen\WObj:=wPaper;
    MoveL Offs(pOrigin,130.36,41.12,6.00),vTravel,z5,tPen\WObj:=wPaper;
    MoveL Offs(pOrigin,130.36,41.12,0.00),v60,z0,tPen\WObj:=wPaper;
    MoveL Offs(pOrigin,129.94,41.55,0.00),v40,z0,tPen\WObj:=wPaper;
    MoveL Offs(pOrigin,130.36,41.12,0.00),v40,fine,tPen\WObj:=wPaper;
    MoveL Offs(pOrigin,130.36,41.12,6.00),v60,z5,tPen\WObj:=wPaper;
    MoveL Offs(pOrigin,133.12,39.85,6.00),vTravel,z5,tPen\WObj:=wPaper;
    MoveL Offs(pOrigin,133.12,39.85,0.00),v60,z0,tPen\WObj:=wPaper;
    MoveL Offs(pOrigin,133.55,39.64,0.00),v40,z0,tPen\WObj:=wPaper;
    MoveL Offs(pOrigin,133.12,39.85,0.00),v40,fine,tPen\WObj:=wPaper;
    MoveL Offs(pOrigin,133.12,39.85,6.00),v60,z5,tPen\WObj:=wPaper;
    MoveL Offs(pOrigin,138.01,42.83,6.00),vTravel,z5,tPen\WObj:=wPaper;
    MoveL Offs(pOrigin,138.01,42.83,0.00),v60,z0,tPen\WObj:=wPaper;
    MoveL Offs(pOrigin,137.80,43.25,0.00),v40,z0,tPen\WObj:=wPaper;
    MoveL Offs(pOrigin,138.01,42.83,0.00),v40,fine,tPen\WObj:=wPaper;
    MoveL Offs(pOrigin,138.01,42.83,6.00),v60,z5,tPen\WObj:=wPaper;
    MoveL Offs(pOrigin,136.74,46.22,6.00),vTravel,z5,tPen\WObj:=wPaper;
    MoveL Offs(pOrigin,136.74,46.22,0.00),v60,z0,tPen\WObj:=wPaper;
    MoveL Offs(pOrigin,137.02,44.95,0.00),v40,z0,tPen\WObj:=wPaper;
    MoveL Offs(pOrigin,138.37,42.40,0.00),v40,z0,tPen\WObj:=wPaper;
    MoveL Offs(pOrigin,140.21,39.85,0.00),v40,z0,tPen\WObj:=wPaper;
    MoveL Offs(pOrigin,141.84,38.36,0.00),v40,fine,tPen\WObj:=wPaper;
    MoveL Offs(pOrigin,141.84,38.36,6.00),v60,z5,tPen\WObj:=wPaper;
    MoveL Offs(pOrigin,136.95,47.50,6.00),vTravel,z5,tPen\WObj:=wPaper;
    MoveL Offs(pOrigin,136.95,47.50,0.00),v60,z0,tPen\WObj:=wPaper;
    MoveL Offs(pOrigin,136.74,47.92,0.00),v40,z0,tPen\WObj:=wPaper;
    MoveL Offs(pOrigin,136.95,47.50,0.00),v40,fine,tPen\WObj:=wPaper;
    MoveL Offs(pOrigin,136.95,47.50,6.00),v60,z5,tPen\WObj:=wPaper;
    MoveL Offs(pOrigin,155.86,38.58,6.00),vTravel,z5,tPen\WObj:=wPaper;
    MoveL Offs(pOrigin,155.86,38.58,0.00),v60,z0,tPen\WObj:=wPaper;
    MoveL Offs(pOrigin,155.65,38.79,0.00),v40,z0,tPen\WObj:=wPaper;
    MoveL Offs(pOrigin,155.86,38.36,0.00),v40,z0,tPen\WObj:=wPaper;
    MoveL Offs(pOrigin,157.14,38.36,0.00),v40,fine,tPen\WObj:=wPaper;
    MoveL Offs(pOrigin,157.14,38.36,6.00),v60,z5,tPen\WObj:=wPaper;
    MoveL Offs(pOrigin,161.81,41.76,6.00),vTravel,z5,tPen\WObj:=wPaper;
    MoveL Offs(pOrigin,161.81,41.76,0.00),v60,z0,tPen\WObj:=wPaper;
    MoveL Offs(pOrigin,161.81,46.86,0.00),v40,z0,tPen\WObj:=wPaper;
    MoveL Offs(pOrigin,162.45,49.62,0.00),v40,fine,tPen\WObj:=wPaper;
    MoveL Offs(pOrigin,162.45,49.62,6.00),v60,z5,tPen\WObj:=wPaper;
    MoveL Offs(pOrigin,159.48,56.42,6.00),vTravel,z5,tPen\WObj:=wPaper;
    MoveL Offs(pOrigin,159.48,56.42,0.00),v60,z0,tPen\WObj:=wPaper;
    MoveL Offs(pOrigin,159.26,56.85,0.00),v40,z0,tPen\WObj:=wPaper;
    MoveL Offs(pOrigin,160.04,58.76,0.00),v40,z0,tPen\WObj:=wPaper;
    MoveL Offs(pOrigin,163.30,64.50,0.00),v40,z0,tPen\WObj:=wPaper;
    MoveL Offs(pOrigin,165.85,66.84,0.00),v40,z0,tPen\WObj:=wPaper;
    MoveL Offs(pOrigin,166.27,67.69,0.00),v40,fine,tPen\WObj:=wPaper;
    MoveL Offs(pOrigin,166.27,67.69,6.00),v60,z5,tPen\WObj:=wPaper;
    MoveL Offs(pOrigin,167.98,65.99,6.00),vTravel,z5,tPen\WObj:=wPaper;
    MoveL Offs(pOrigin,167.98,65.99,0.00),v60,z0,tPen\WObj:=wPaper;
    MoveL Offs(pOrigin,165.57,62.38,0.00),v40,z0,tPen\WObj:=wPaper;
    MoveL Offs(pOrigin,164.79,60.04,0.00),v40,fine,tPen\WObj:=wPaper;
    MoveL Offs(pOrigin,164.79,60.04,6.00),v60,z5,tPen\WObj:=wPaper;
    MoveL Offs(pOrigin,163.51,64.93,6.00),vTravel,z5,tPen\WObj:=wPaper;
    MoveL Offs(pOrigin,163.51,64.93,0.00),v60,z0,tPen\WObj:=wPaper;
    MoveL Offs(pOrigin,164.36,65.78,0.00),v40,z0,tPen\WObj:=wPaper;
    MoveL Offs(pOrigin,163.51,64.93,0.00),v40,fine,tPen\WObj:=wPaper;
    MoveL Offs(pOrigin,163.51,64.93,6.00),v60,z5,tPen\WObj:=wPaper;
    MoveL Offs(pOrigin,161.81,69.81,6.00),vTravel,z5,tPen\WObj:=wPaper;
    MoveL Offs(pOrigin,161.81,69.81,0.00),v60,z0,tPen\WObj:=wPaper;
    MoveL Offs(pOrigin,159.90,70.24,0.00),v40,z0,tPen\WObj:=wPaper;
    MoveL Offs(pOrigin,156.93,70.24,0.00),v40,z0,tPen\WObj:=wPaper;
  ENDPROC

  PROC DrawPart99()
    MoveL Offs(pOrigin,156.07,69.39,0.00),v40,z0,tPen\WObj:=wPaper;
    MoveL Offs(pOrigin,156.07,69.39,0.00),v40,z0,tPen\WObj:=wPaper;
    MoveL Offs(pOrigin,155.01,68.47,0.00),v40,z0,tPen\WObj:=wPaper;
    MoveL Offs(pOrigin,152.89,67.90,0.00),v40,z0,tPen\WObj:=wPaper;
    MoveL Offs(pOrigin,152.60,68.11,0.00),v40,z0,tPen\WObj:=wPaper;
    MoveL Offs(pOrigin,153.31,69.32,0.00),v40,z0,tPen\WObj:=wPaper;
    MoveL Offs(pOrigin,154.80,69.81,0.00),v40,z0,tPen\WObj:=wPaper;
    MoveL Offs(pOrigin,156.07,69.81,0.00),v40,fine,tPen\WObj:=wPaper;
    MoveL Offs(pOrigin,156.07,69.81,6.00),v60,z5,tPen\WObj:=wPaper;
    MoveL Offs(pOrigin,157.14,79.80,6.00),vTravel,z5,tPen\WObj:=wPaper;
    MoveL Offs(pOrigin,157.14,79.80,0.00),v60,z0,tPen\WObj:=wPaper;
    MoveL Offs(pOrigin,156.36,81.50,0.00),v40,z0,tPen\WObj:=wPaper;
    MoveL Offs(pOrigin,153.52,85.32,0.00),v40,z0,tPen\WObj:=wPaper;
    MoveL Offs(pOrigin,149.49,89.36,0.00),v40,fine,tPen\WObj:=wPaper;
    MoveL Offs(pOrigin,149.49,89.36,6.00),v60,z5,tPen\WObj:=wPaper;
    MoveL Offs(pOrigin,148.43,90.43,6.00),vTravel,z5,tPen\WObj:=wPaper;
    MoveL Offs(pOrigin,148.43,90.43,0.00),v60,z0,tPen\WObj:=wPaper;
    MoveL Offs(pOrigin,148.21,91.06,0.00),v40,z0,tPen\WObj:=wPaper;
    MoveL Offs(pOrigin,147.15,91.28,0.00),v40,z0,tPen\WObj:=wPaper;
    MoveL Offs(pOrigin,147.15,91.28,0.00),v40,z0,tPen\WObj:=wPaper;
    MoveL Offs(pOrigin,147.15,90.64,0.00),v40,z0,tPen\WObj:=wPaper;
    MoveL Offs(pOrigin,147.57,90.21,0.00),v40,z0,tPen\WObj:=wPaper;
    MoveL Offs(pOrigin,148.21,90.21,0.00),v40,z0,tPen\WObj:=wPaper;
    MoveL Offs(pOrigin,148.21,90.21,0.00),v40,z0,tPen\WObj:=wPaper;
    MoveL Offs(pOrigin,148.43,89.57,0.00),v40,z0,tPen\WObj:=wPaper;
    MoveL Offs(pOrigin,149.27,89.43,0.00),v40,z0,tPen\WObj:=wPaper;
    MoveL Offs(pOrigin,149.20,90.14,0.00),v40,z0,tPen\WObj:=wPaper;
    MoveL Offs(pOrigin,148.43,90.43,0.00),v40,fine,tPen\WObj:=wPaper;
    MoveL Offs(pOrigin,148.43,90.43,6.00),v60,z5,tPen\WObj:=wPaper;
    MoveL Offs(pOrigin,147.15,91.28,6.00),vTravel,z5,tPen\WObj:=wPaper;
    MoveL Offs(pOrigin,147.15,91.28,0.00),v60,z0,tPen\WObj:=wPaper;
    MoveL Offs(pOrigin,146.73,91.28,0.00),v40,z0,tPen\WObj:=wPaper;
    MoveL Offs(pOrigin,146.51,91.70,0.00),v40,z0,tPen\WObj:=wPaper;
    MoveL Offs(pOrigin,146.73,91.49,0.00),v40,fine,tPen\WObj:=wPaper;
    MoveL Offs(pOrigin,146.73,91.49,6.00),v60,z5,tPen\WObj:=wPaper;
    MoveL Offs(pOrigin,143.32,90.21,6.00),vTravel,z5,tPen\WObj:=wPaper;
    MoveL Offs(pOrigin,143.32,90.21,0.00),v60,z0,tPen\WObj:=wPaper;
    MoveL Offs(pOrigin,150.55,83.41,0.00),v40,z0,tPen\WObj:=wPaper;
    MoveL Offs(pOrigin,152.89,80.86,0.00),v40,z0,tPen\WObj:=wPaper;
    MoveL Offs(pOrigin,153.10,80.01,0.00),v40,fine,tPen\WObj:=wPaper;
    MoveL Offs(pOrigin,153.10,80.01,6.00),v60,z5,tPen\WObj:=wPaper;
    MoveL Offs(pOrigin,151.61,81.93,6.00),vTravel,z5,tPen\WObj:=wPaper;
    MoveL Offs(pOrigin,151.61,81.93,0.00),v60,z0,tPen\WObj:=wPaper;
    MoveL Offs(pOrigin,150.98,82.56,0.00),v40,z0,tPen\WObj:=wPaper;
    MoveL Offs(pOrigin,151.61,81.93,0.00),v40,fine,tPen\WObj:=wPaper;
    MoveL Offs(pOrigin,151.61,81.93,6.00),v60,z5,tPen\WObj:=wPaper;
    MoveL Offs(pOrigin,150.05,83.77,6.00),vTravel,z5,tPen\WObj:=wPaper;
    MoveL Offs(pOrigin,150.05,83.77,0.00),v60,z0,tPen\WObj:=wPaper;
    MoveL Offs(pOrigin,146.09,87.66,0.00),v40,z0,tPen\WObj:=wPaper;
    MoveL Offs(pOrigin,150.05,83.77,0.00),v40,fine,tPen\WObj:=wPaper;
    MoveL Offs(pOrigin,150.05,83.77,6.00),v60,z5,tPen\WObj:=wPaper;
    MoveL Offs(pOrigin,148.43,81.50,6.00),vTravel,z5,tPen\WObj:=wPaper;
    MoveL Offs(pOrigin,148.43,81.50,0.00),v60,z0,tPen\WObj:=wPaper;
    MoveL Offs(pOrigin,148.85,81.29,0.00),v40,z0,tPen\WObj:=wPaper;
    MoveL Offs(pOrigin,148.43,81.50,0.00),v40,z0,tPen\WObj:=wPaper;
    MoveL Offs(pOrigin,149.27,81.07,0.00),v40,z0,tPen\WObj:=wPaper;
    MoveL Offs(pOrigin,149.70,80.86,0.00),v40,z0,tPen\WObj:=wPaper;
    MoveL Offs(pOrigin,149.27,81.07,0.00),v40,fine,tPen\WObj:=wPaper;
    MoveL Offs(pOrigin,149.27,81.07,6.00),v60,z5,tPen\WObj:=wPaper;
    MoveL Offs(pOrigin,153.52,85.11,6.00),vTravel,z5,tPen\WObj:=wPaper;
    MoveL Offs(pOrigin,153.52,85.11,0.00),v60,z0,tPen\WObj:=wPaper;
    MoveL Offs(pOrigin,152.46,86.18,0.00),v40,z0,tPen\WObj:=wPaper;
    MoveL Offs(pOrigin,153.52,85.11,0.00),v40,fine,tPen\WObj:=wPaper;
    MoveL Offs(pOrigin,153.52,85.11,6.00),v60,z5,tPen\WObj:=wPaper;
    MoveL Offs(pOrigin,152.04,86.81,6.00),vTravel,z5,tPen\WObj:=wPaper;
    MoveL Offs(pOrigin,152.04,86.81,0.00),v60,z0,tPen\WObj:=wPaper;
    MoveL Offs(pOrigin,150.55,88.30,0.00),v40,z0,tPen\WObj:=wPaper;
    MoveL Offs(pOrigin,152.04,86.81,0.00),v40,fine,tPen\WObj:=wPaper;
    MoveL Offs(pOrigin,152.04,86.81,6.00),v60,z5,tPen\WObj:=wPaper;
    MoveL Offs(pOrigin,154.38,92.97,6.00),vTravel,z5,tPen\WObj:=wPaper;
    MoveL Offs(pOrigin,154.38,92.97,0.00),v60,z0,tPen\WObj:=wPaper;
    MoveL Offs(pOrigin,152.89,93.61,0.00),v40,z0,tPen\WObj:=wPaper;
    MoveL Offs(pOrigin,152.68,94.04,0.00),v40,z0,tPen\WObj:=wPaper;
    MoveL Offs(pOrigin,152.89,93.82,0.00),v40,fine,tPen\WObj:=wPaper;
    MoveL Offs(pOrigin,152.89,93.82,6.00),v60,z5,tPen\WObj:=wPaper;
    MoveL Offs(pOrigin,160.54,93.61,6.00),vTravel,z5,tPen\WObj:=wPaper;
    MoveL Offs(pOrigin,160.54,93.61,0.00),v60,z0,tPen\WObj:=wPaper;
    MoveL Offs(pOrigin,160.75,94.04,0.00),v40,z0,tPen\WObj:=wPaper;
    MoveL Offs(pOrigin,160.54,93.61,0.00),v40,fine,tPen\WObj:=wPaper;
    MoveL Offs(pOrigin,160.54,93.61,6.00),v60,z5,tPen\WObj:=wPaper;
    MoveL Offs(pOrigin,162.45,92.12,6.00),vTravel,z5,tPen\WObj:=wPaper;
    MoveL Offs(pOrigin,162.45,92.12,0.00),v60,z0,tPen\WObj:=wPaper;
    MoveL Offs(pOrigin,162.31,91.70,0.00),v40,z0,tPen\WObj:=wPaper;
    MoveL Offs(pOrigin,162.88,90.85,0.00),v40,z0,tPen\WObj:=wPaper;
    MoveL Offs(pOrigin,165.21,82.14,0.00),v40,z0,tPen\WObj:=wPaper;
    MoveL Offs(pOrigin,167.98,75.55,0.00),v40,z0,tPen\WObj:=wPaper;
    MoveL Offs(pOrigin,167.76,74.70,0.00),v40,z0,tPen\WObj:=wPaper;
    MoveL Offs(pOrigin,160.11,77.32,0.00),v40,z0,tPen\WObj:=wPaper;
    MoveL Offs(pOrigin,159.83,77.68,0.00),v40,z0,tPen\WObj:=wPaper;
    MoveL Offs(pOrigin,161.39,82.99,0.00),v40,z0,tPen\WObj:=wPaper;
    MoveL Offs(pOrigin,162.24,91.49,0.00),v40,fine,tPen\WObj:=wPaper;
    MoveL Offs(pOrigin,162.24,91.49,6.00),v60,z5,tPen\WObj:=wPaper;
    MoveL Offs(pOrigin,163.73,92.55,6.00),vTravel,z5,tPen\WObj:=wPaper;
    MoveL Offs(pOrigin,163.73,92.55,0.00),v60,z0,tPen\WObj:=wPaper;
    MoveL Offs(pOrigin,163.30,94.46,0.00),v40,z0,tPen\WObj:=wPaper;
    MoveL Offs(pOrigin,163.94,95.67,0.00),v40,z0,tPen\WObj:=wPaper;
    MoveL Offs(pOrigin,164.65,95.31,0.00),v40,z0,tPen\WObj:=wPaper;
    MoveL Offs(pOrigin,165.14,93.61,0.00),v40,z0,tPen\WObj:=wPaper;
    MoveL Offs(pOrigin,167.34,90.64,0.00),v40,z0,tPen\WObj:=wPaper;
    MoveL Offs(pOrigin,177.18,81.36,0.00),v40,z0,tPen\WObj:=wPaper;
    MoveL Offs(pOrigin,163.73,92.55,0.00),v40,fine,tPen\WObj:=wPaper;
    MoveL Offs(pOrigin,163.73,92.55,6.00),v60,z5,tPen\WObj:=wPaper;
    MoveL Offs(pOrigin,165.64,92.55,6.00),vTravel,z5,tPen\WObj:=wPaper;
    MoveL Offs(pOrigin,165.64,92.55,0.00),v60,z0,tPen\WObj:=wPaper;
    MoveL Offs(pOrigin,165.21,93.19,0.00),v40,z0,tPen\WObj:=wPaper;
    MoveL Offs(pOrigin,165.64,92.55,0.00),v40,fine,tPen\WObj:=wPaper;
    MoveL Offs(pOrigin,165.64,92.55,6.00),v60,z5,tPen\WObj:=wPaper;
    MoveL Offs(pOrigin,166.70,91.49,6.00),vTravel,z5,tPen\WObj:=wPaper;
    MoveL Offs(pOrigin,166.70,91.49,0.00),v60,z0,tPen\WObj:=wPaper;
    MoveL Offs(pOrigin,166.27,91.91,0.00),v40,z0,tPen\WObj:=wPaper;
    MoveL Offs(pOrigin,166.70,91.49,0.00),v40,fine,tPen\WObj:=wPaper;
    MoveL Offs(pOrigin,166.70,91.49,6.00),v60,z5,tPen\WObj:=wPaper;
    MoveL Offs(pOrigin,167.76,90.00,6.00),vTravel,z5,tPen\WObj:=wPaper;
    MoveL Offs(pOrigin,167.76,90.00,0.00),v60,z0,tPen\WObj:=wPaper;
    MoveL Offs(pOrigin,167.12,90.64,0.00),v40,z0,tPen\WObj:=wPaper;
    MoveL Offs(pOrigin,167.76,90.00,0.00),v40,fine,tPen\WObj:=wPaper;
    MoveL Offs(pOrigin,167.76,90.00,6.00),v60,z5,tPen\WObj:=wPaper;
    MoveL Offs(pOrigin,169.46,88.30,6.00),vTravel,z5,tPen\WObj:=wPaper;
    MoveL Offs(pOrigin,169.46,88.30,0.00),v60,z0,tPen\WObj:=wPaper;
    MoveL Offs(pOrigin,167.98,89.79,0.00),v40,z0,tPen\WObj:=wPaper;
  ENDPROC

  PROC DrawPart100()
    MoveL Offs(pOrigin,169.46,88.30,0.00),v40,fine,tPen\WObj:=wPaper;
    MoveL Offs(pOrigin,169.46,88.30,6.00),v60,z5,tPen\WObj:=wPaper;
    MoveL Offs(pOrigin,170.31,87.45,6.00),vTravel,z5,tPen\WObj:=wPaper;
    MoveL Offs(pOrigin,170.31,87.45,0.00),v60,z0,tPen\WObj:=wPaper;
    MoveL Offs(pOrigin,169.68,88.09,0.00),v40,z0,tPen\WObj:=wPaper;
    MoveL Offs(pOrigin,170.31,87.45,0.00),v40,fine,tPen\WObj:=wPaper;
    MoveL Offs(pOrigin,170.31,87.45,6.00),v60,z5,tPen\WObj:=wPaper;
    MoveL Offs(pOrigin,172.65,85.32,6.00),vTravel,z5,tPen\WObj:=wPaper;
    MoveL Offs(pOrigin,172.65,85.32,0.00),v60,z0,tPen\WObj:=wPaper;
    MoveL Offs(pOrigin,170.95,87.03,0.00),v40,z0,tPen\WObj:=wPaper;
    MoveL Offs(pOrigin,172.65,85.32,0.00),v40,fine,tPen\WObj:=wPaper;
    MoveL Offs(pOrigin,172.65,85.32,6.00),v60,z5,tPen\WObj:=wPaper;
    MoveL Offs(pOrigin,174.35,83.84,6.00),vTravel,z5,tPen\WObj:=wPaper;
    MoveL Offs(pOrigin,174.35,83.84,0.00),v60,z0,tPen\WObj:=wPaper;
    MoveL Offs(pOrigin,173.29,84.90,0.00),v40,z0,tPen\WObj:=wPaper;
    MoveL Offs(pOrigin,174.35,83.84,0.00),v40,fine,tPen\WObj:=wPaper;
    MoveL Offs(pOrigin,174.35,83.84,6.00),v60,z5,tPen\WObj:=wPaper;
    MoveL Offs(pOrigin,175.20,86.81,6.00),vTravel,z5,tPen\WObj:=wPaper;
    MoveL Offs(pOrigin,175.20,86.81,0.00),v60,z0,tPen\WObj:=wPaper;
    MoveL Offs(pOrigin,176.83,86.32,0.00),v40,z0,tPen\WObj:=wPaper;
    MoveL Offs(pOrigin,177.32,85.11,0.00),v40,z0,tPen\WObj:=wPaper;
    MoveL Offs(pOrigin,177.32,85.11,0.00),v40,z0,tPen\WObj:=wPaper;
    MoveL Offs(pOrigin,178.60,84.76,0.00),v40,z0,tPen\WObj:=wPaper;
    MoveL Offs(pOrigin,179.24,83.70,0.00),v40,z0,tPen\WObj:=wPaper;
    MoveL Offs(pOrigin,180.87,82.70,0.00),v40,z0,tPen\WObj:=wPaper;
    MoveL Offs(pOrigin,181.15,81.93,0.00),v40,fine,tPen\WObj:=wPaper;
    MoveL Offs(pOrigin,181.15,81.93,6.00),v60,z5,tPen\WObj:=wPaper;
    MoveL Offs(pOrigin,181.15,80.65,6.00),vTravel,z5,tPen\WObj:=wPaper;
    MoveL Offs(pOrigin,181.15,80.65,0.00),v60,z0,tPen\WObj:=wPaper;
    MoveL Offs(pOrigin,181.36,80.01,0.00),v40,z0,tPen\WObj:=wPaper;
    MoveL Offs(pOrigin,183.27,78.45,0.00),v40,z0,tPen\WObj:=wPaper;
    MoveL Offs(pOrigin,184.55,77.89,0.00),v40,z0,tPen\WObj:=wPaper;
    MoveL Offs(pOrigin,185.61,78.31,0.00),v40,fine,tPen\WObj:=wPaper;
    MoveL Offs(pOrigin,185.61,78.31,6.00),v60,z5,tPen\WObj:=wPaper;
    MoveL Offs(pOrigin,179.80,78.53,6.00),vTravel,z5,tPen\WObj:=wPaper;
    MoveL Offs(pOrigin,179.80,78.53,0.00),v60,z0,tPen\WObj:=wPaper;
    MoveL Offs(pOrigin,179.80,79.16,0.00),v40,z0,tPen\WObj:=wPaper;
    MoveL Offs(pOrigin,177.61,81.15,0.00),v40,z0,tPen\WObj:=wPaper;
    MoveL Offs(pOrigin,165.21,86.18,0.00),v40,z0,tPen\WObj:=wPaper;
    MoveL Offs(pOrigin,167.05,80.44,0.00),v40,z0,tPen\WObj:=wPaper;
    MoveL Offs(pOrigin,169.60,74.91,0.00),v40,z0,tPen\WObj:=wPaper;
    MoveL Offs(pOrigin,170.74,73.28,0.00),v40,z0,tPen\WObj:=wPaper;
    MoveL Offs(pOrigin,171.80,73.43,0.00),v40,z0,tPen\WObj:=wPaper;
    MoveL Offs(pOrigin,176.26,77.32,0.00),v40,z0,tPen\WObj:=wPaper;
    MoveL Offs(pOrigin,179.80,78.53,0.00),v40,z0,tPen\WObj:=wPaper;
    MoveL Offs(pOrigin,179.66,79.16,0.00),v40,z0,tPen\WObj:=wPaper;
    MoveL Offs(pOrigin,179.45,79.59,0.00),v40,z0,tPen\WObj:=wPaper;
    MoveL Offs(pOrigin,179.66,79.16,0.00),v40,fine,tPen\WObj:=wPaper;
    MoveL Offs(pOrigin,179.66,79.16,6.00),v60,z5,tPen\WObj:=wPaper;
    MoveL Offs(pOrigin,178.81,80.22,6.00),vTravel,z5,tPen\WObj:=wPaper;
    MoveL Offs(pOrigin,178.81,80.22,0.00),v60,z0,tPen\WObj:=wPaper;
    MoveL Offs(pOrigin,179.02,79.80,0.00),v40,z0,tPen\WObj:=wPaper;
    MoveL Offs(pOrigin,178.81,80.22,0.00),v40,fine,tPen\WObj:=wPaper;
    MoveL Offs(pOrigin,178.81,80.22,6.00),v60,z5,tPen\WObj:=wPaper;
    MoveL Offs(pOrigin,179.02,81.71,6.00),vTravel,z5,tPen\WObj:=wPaper;
    MoveL Offs(pOrigin,179.02,81.71,0.00),v60,z0,tPen\WObj:=wPaper;
    MoveL Offs(pOrigin,178.60,82.14,0.00),v40,z0,tPen\WObj:=wPaper;
    MoveL Offs(pOrigin,179.02,81.71,0.00),v40,z0,tPen\WObj:=wPaper;
    MoveL Offs(pOrigin,179.66,81.71,0.00),v40,z0,tPen\WObj:=wPaper;
    MoveL Offs(pOrigin,179.88,82.99,0.00),v40,fine,tPen\WObj:=wPaper;
    MoveL Offs(pOrigin,179.88,82.99,6.00),v60,z5,tPen\WObj:=wPaper;
    MoveL Offs(pOrigin,173.93,87.66,6.00),vTravel,z5,tPen\WObj:=wPaper;
    MoveL Offs(pOrigin,173.93,87.66,0.00),v60,z0,tPen\WObj:=wPaper;
    MoveL Offs(pOrigin,172.86,88.72,0.00),v40,z0,tPen\WObj:=wPaper;
    MoveL Offs(pOrigin,173.93,87.66,0.00),v40,fine,tPen\WObj:=wPaper;
    MoveL Offs(pOrigin,173.93,87.66,6.00),v60,z5,tPen\WObj:=wPaper;
    MoveL Offs(pOrigin,170.31,90.85,6.00),vTravel,z5,tPen\WObj:=wPaper;
    MoveL Offs(pOrigin,170.31,90.85,0.00),v60,z0,tPen\WObj:=wPaper;
    MoveL Offs(pOrigin,168.82,91.28,0.00),v40,z0,tPen\WObj:=wPaper;
    MoveL Offs(pOrigin,168.12,92.34,0.00),v40,z0,tPen\WObj:=wPaper;
    MoveL Offs(pOrigin,167.98,93.40,0.00),v40,z0,tPen\WObj:=wPaper;
    MoveL Offs(pOrigin,167.98,94.46,0.00),v40,z0,tPen\WObj:=wPaper;
    MoveL Offs(pOrigin,167.12,94.53,0.00),v40,z0,tPen\WObj:=wPaper;
    MoveL Offs(pOrigin,166.77,94.89,0.00),v40,z0,tPen\WObj:=wPaper;
    MoveL Offs(pOrigin,167.12,95.95,0.00),v40,z0,tPen\WObj:=wPaper;
    MoveL Offs(pOrigin,168.40,96.38,0.00),v40,z0,tPen\WObj:=wPaper;
    MoveL Offs(pOrigin,168.82,95.53,0.00),v40,fine,tPen\WObj:=wPaper;
    MoveL Offs(pOrigin,168.82,95.53,6.00),v60,z5,tPen\WObj:=wPaper;
    MoveL Offs(pOrigin,173.29,96.59,6.00),vTravel,z5,tPen\WObj:=wPaper;
    MoveL Offs(pOrigin,173.29,96.59,0.00),v60,z0,tPen\WObj:=wPaper;
    MoveL Offs(pOrigin,180.51,104.24,0.00),v40,z0,tPen\WObj:=wPaper;
    MoveL Offs(pOrigin,193.05,116.56,0.00),v40,fine,tPen\WObj:=wPaper;
    MoveL Offs(pOrigin,193.05,116.56,6.00),v60,z5,tPen\WObj:=wPaper;
    MoveL Offs(pOrigin,193.69,114.22,6.00),vTravel,z5,tPen\WObj:=wPaper;
    MoveL Offs(pOrigin,193.69,114.22,0.00),v60,z0,tPen\WObj:=wPaper;
    MoveL Offs(pOrigin,194.11,114.65,0.00),v40,z0,tPen\WObj:=wPaper;
    MoveL Offs(pOrigin,193.69,114.22,0.00),v40,fine,tPen\WObj:=wPaper;
    MoveL Offs(pOrigin,193.69,114.22,6.00),v60,z5,tPen\WObj:=wPaper;
    MoveL Offs(pOrigin,191.99,112.74,6.00),vTravel,z5,tPen\WObj:=wPaper;
    MoveL Offs(pOrigin,191.99,112.74,0.00),v60,z0,tPen\WObj:=wPaper;
    MoveL Offs(pOrigin,192.84,113.59,0.00),v40,z0,tPen\WObj:=wPaper;
    MoveL Offs(pOrigin,191.99,112.74,0.00),v40,fine,tPen\WObj:=wPaper;
    MoveL Offs(pOrigin,191.99,112.74,6.00),v60,z5,tPen\WObj:=wPaper;
    MoveL Offs(pOrigin,190.50,111.25,6.00),vTravel,z5,tPen\WObj:=wPaper;
    MoveL Offs(pOrigin,190.50,111.25,0.00),v60,z0,tPen\WObj:=wPaper;
    MoveL Offs(pOrigin,191.35,112.10,0.00),v40,z0,tPen\WObj:=wPaper;
    MoveL Offs(pOrigin,190.50,111.25,0.00),v40,fine,tPen\WObj:=wPaper;
    MoveL Offs(pOrigin,190.50,111.25,6.00),v60,z5,tPen\WObj:=wPaper;
    MoveL Offs(pOrigin,188.16,108.70,6.00),vTravel,z5,tPen\WObj:=wPaper;
    MoveL Offs(pOrigin,188.16,108.70,0.00),v60,z0,tPen\WObj:=wPaper;
    MoveL Offs(pOrigin,188.59,109.12,0.00),v40,z0,tPen\WObj:=wPaper;
    MoveL Offs(pOrigin,188.16,108.70,0.00),v40,fine,tPen\WObj:=wPaper;
    MoveL Offs(pOrigin,188.16,108.70,6.00),v60,z5,tPen\WObj:=wPaper;
    MoveL Offs(pOrigin,186.46,109.97,6.00),vTravel,z5,tPen\WObj:=wPaper;
    MoveL Offs(pOrigin,186.46,109.97,0.00),v60,z0,tPen\WObj:=wPaper;
    MoveL Offs(pOrigin,186.89,110.40,0.00),v40,z0,tPen\WObj:=wPaper;
    MoveL Offs(pOrigin,186.46,109.97,0.00),v40,fine,tPen\WObj:=wPaper;
    MoveL Offs(pOrigin,186.46,109.97,6.00),v60,z5,tPen\WObj:=wPaper;
    MoveL Offs(pOrigin,184.76,108.28,6.00),vTravel,z5,tPen\WObj:=wPaper;
    MoveL Offs(pOrigin,184.76,108.28,0.00),v60,z0,tPen\WObj:=wPaper;
    MoveL Offs(pOrigin,186.25,109.76,0.00),v40,z0,tPen\WObj:=wPaper;
    MoveL Offs(pOrigin,184.76,108.28,0.00),v40,fine,tPen\WObj:=wPaper;
    MoveL Offs(pOrigin,184.76,108.28,6.00),v60,z5,tPen\WObj:=wPaper;
    MoveL Offs(pOrigin,183.70,107.21,6.00),vTravel,z5,tPen\WObj:=wPaper;
    MoveL Offs(pOrigin,183.70,107.21,0.00),v60,z0,tPen\WObj:=wPaper;
    MoveL Offs(pOrigin,184.55,108.06,0.00),v40,z0,tPen\WObj:=wPaper;
    MoveL Offs(pOrigin,183.70,107.21,0.00),v40,fine,tPen\WObj:=wPaper;
    MoveL Offs(pOrigin,183.70,107.21,6.00),v60,z5,tPen\WObj:=wPaper;
    MoveL Offs(pOrigin,182.21,105.72,6.00),vTravel,z5,tPen\WObj:=wPaper;
    MoveL Offs(pOrigin,182.21,105.72,0.00),v60,z0,tPen\WObj:=wPaper;
  ENDPROC

  PROC DrawPart101()
    MoveL Offs(pOrigin,183.06,106.57,0.00),v40,z0,tPen\WObj:=wPaper;
    MoveL Offs(pOrigin,182.21,105.72,0.00),v40,fine,tPen\WObj:=wPaper;
    MoveL Offs(pOrigin,182.21,105.72,6.00),v60,z5,tPen\WObj:=wPaper;
    MoveL Offs(pOrigin,181.15,104.66,6.00),vTravel,z5,tPen\WObj:=wPaper;
    MoveL Offs(pOrigin,181.15,104.66,0.00),v60,z0,tPen\WObj:=wPaper;
    MoveL Offs(pOrigin,182.00,105.51,0.00),v40,z0,tPen\WObj:=wPaper;
    MoveL Offs(pOrigin,181.15,104.66,0.00),v40,fine,tPen\WObj:=wPaper;
    MoveL Offs(pOrigin,181.15,104.66,6.00),v60,z5,tPen\WObj:=wPaper;
    MoveL Offs(pOrigin,176.90,100.20,6.00),vTravel,z5,tPen\WObj:=wPaper;
    MoveL Offs(pOrigin,176.90,100.20,0.00),v60,z0,tPen\WObj:=wPaper;
    MoveL Offs(pOrigin,177.54,100.84,0.00),v40,z0,tPen\WObj:=wPaper;
    MoveL Offs(pOrigin,176.90,100.20,0.00),v40,fine,tPen\WObj:=wPaper;
    MoveL Offs(pOrigin,176.90,100.20,6.00),v60,z5,tPen\WObj:=wPaper;
    MoveL Offs(pOrigin,175.84,99.14,6.00),vTravel,z5,tPen\WObj:=wPaper;
    MoveL Offs(pOrigin,175.84,99.14,0.00),v60,z0,tPen\WObj:=wPaper;
    MoveL Offs(pOrigin,176.26,99.56,0.00),v40,z0,tPen\WObj:=wPaper;
    MoveL Offs(pOrigin,175.84,99.14,0.00),v40,fine,tPen\WObj:=wPaper;
    MoveL Offs(pOrigin,175.84,99.14,6.00),v60,z5,tPen\WObj:=wPaper;
    MoveL Offs(pOrigin,174.35,97.65,6.00),vTravel,z5,tPen\WObj:=wPaper;
    MoveL Offs(pOrigin,174.35,97.65,0.00),v60,z0,tPen\WObj:=wPaper;
    MoveL Offs(pOrigin,175.20,98.50,0.00),v40,z0,tPen\WObj:=wPaper;
    MoveL Offs(pOrigin,174.35,97.65,0.00),v40,fine,tPen\WObj:=wPaper;
    MoveL Offs(pOrigin,174.35,97.65,6.00),v60,z5,tPen\WObj:=wPaper;
    MoveL Offs(pOrigin,174.99,94.46,6.00),vTravel,z5,tPen\WObj:=wPaper;
    MoveL Offs(pOrigin,174.99,94.46,0.00),v60,z0,tPen\WObj:=wPaper;
    MoveL Offs(pOrigin,174.35,95.10,0.00),v40,z0,tPen\WObj:=wPaper;
    MoveL Offs(pOrigin,174.99,94.46,0.00),v40,fine,tPen\WObj:=wPaper;
    MoveL Offs(pOrigin,174.99,94.46,6.00),v60,z5,tPen\WObj:=wPaper;
    MoveL Offs(pOrigin,176.05,93.61,6.00),vTravel,z5,tPen\WObj:=wPaper;
    MoveL Offs(pOrigin,176.05,93.61,0.00),v60,z0,tPen\WObj:=wPaper;
    MoveL Offs(pOrigin,175.41,94.25,0.00),v40,z0,tPen\WObj:=wPaper;
    MoveL Offs(pOrigin,176.05,93.61,0.00),v40,z0,tPen\WObj:=wPaper;
    MoveL Offs(pOrigin,176.90,92.97,0.00),v40,z0,tPen\WObj:=wPaper;
    MoveL Offs(pOrigin,176.48,93.40,0.00),v40,z0,tPen\WObj:=wPaper;
    MoveL Offs(pOrigin,176.90,92.97,0.00),v40,fine,tPen\WObj:=wPaper;
    MoveL Offs(pOrigin,176.90,92.97,6.00),v60,z5,tPen\WObj:=wPaper;
    MoveL Offs(pOrigin,165.00,87.24,6.00),vTravel,z5,tPen\WObj:=wPaper;
    MoveL Offs(pOrigin,165.00,87.24,0.00),v60,z0,tPen\WObj:=wPaper;
    MoveL Offs(pOrigin,165.00,86.60,0.00),v40,z0,tPen\WObj:=wPaper;
    MoveL Offs(pOrigin,165.00,87.24,0.00),v40,z0,tPen\WObj:=wPaper;
    MoveL Offs(pOrigin,164.79,87.66,0.00),v40,z0,tPen\WObj:=wPaper;
    MoveL Offs(pOrigin,163.94,91.91,0.00),v40,z0,tPen\WObj:=wPaper;
    MoveL Offs(pOrigin,164.79,87.66,0.00),v40,fine,tPen\WObj:=wPaper;
    MoveL Offs(pOrigin,164.79,87.66,6.00),v60,z5,tPen\WObj:=wPaper;
    MoveL Offs(pOrigin,166.27,75.34,6.00),vTravel,z5,tPen\WObj:=wPaper;
    MoveL Offs(pOrigin,166.27,75.34,0.00),v60,z0,tPen\WObj:=wPaper;
    MoveL Offs(pOrigin,166.70,75.12,0.00),v40,z0,tPen\WObj:=wPaper;
    MoveL Offs(pOrigin,166.27,75.34,0.00),v40,fine,tPen\WObj:=wPaper;
    MoveL Offs(pOrigin,166.27,75.34,6.00),v60,z5,tPen\WObj:=wPaper;
    MoveL Offs(pOrigin,166.91,73.43,6.00),vTravel,z5,tPen\WObj:=wPaper;
    MoveL Offs(pOrigin,166.91,73.43,0.00),v60,z0,tPen\WObj:=wPaper;
    MoveL Offs(pOrigin,167.34,73.21,0.00),v40,z0,tPen\WObj:=wPaper;
    MoveL Offs(pOrigin,166.91,73.43,0.00),v40,fine,tPen\WObj:=wPaper;
    MoveL Offs(pOrigin,166.91,73.43,6.00),v60,z5,tPen\WObj:=wPaper;
    MoveL Offs(pOrigin,168.61,72.57,6.00),vTravel,z5,tPen\WObj:=wPaper;
    MoveL Offs(pOrigin,168.61,72.57,0.00),v60,z0,tPen\WObj:=wPaper;
    MoveL Offs(pOrigin,169.04,72.36,0.00),v40,z0,tPen\WObj:=wPaper;
    MoveL Offs(pOrigin,168.61,72.57,0.00),v40,fine,tPen\WObj:=wPaper;
    MoveL Offs(pOrigin,168.61,72.57,6.00),v60,z5,tPen\WObj:=wPaper;
    MoveL Offs(pOrigin,170.52,73.21,6.00),vTravel,z5,tPen\WObj:=wPaper;
    MoveL Offs(pOrigin,170.52,73.21,0.00),v60,z0,tPen\WObj:=wPaper;
    MoveL Offs(pOrigin,170.10,73.64,0.00),v40,z0,tPen\WObj:=wPaper;
    MoveL Offs(pOrigin,170.52,73.21,0.00),v40,fine,tPen\WObj:=wPaper;
    MoveL Offs(pOrigin,170.52,73.21,6.00),v60,z5,tPen\WObj:=wPaper;
    MoveL Offs(pOrigin,169.46,74.91,6.00),vTravel,z5,tPen\WObj:=wPaper;
    MoveL Offs(pOrigin,169.46,74.91,0.00),v60,z0,tPen\WObj:=wPaper;
    MoveL Offs(pOrigin,169.25,75.34,0.00),v40,z0,tPen\WObj:=wPaper;
    MoveL Offs(pOrigin,169.46,74.91,0.00),v40,fine,tPen\WObj:=wPaper;
    MoveL Offs(pOrigin,169.46,74.91,6.00),v60,z5,tPen\WObj:=wPaper;
    MoveL Offs(pOrigin,173.07,74.49,6.00),vTravel,z5,tPen\WObj:=wPaper;
    MoveL Offs(pOrigin,173.07,74.49,0.00),v60,z0,tPen\WObj:=wPaper;
    MoveL Offs(pOrigin,173.50,74.91,0.00),v40,z0,tPen\WObj:=wPaper;
    MoveL Offs(pOrigin,173.07,74.49,0.00),v40,fine,tPen\WObj:=wPaper;
    MoveL Offs(pOrigin,173.07,74.49,6.00),v60,z5,tPen\WObj:=wPaper;
    MoveL Offs(pOrigin,173.93,73.21,6.00),vTravel,z5,tPen\WObj:=wPaper;
    MoveL Offs(pOrigin,173.93,73.21,0.00),v60,z0,tPen\WObj:=wPaper;
    MoveL Offs(pOrigin,174.77,74.06,0.00),v40,z0,tPen\WObj:=wPaper;
    MoveL Offs(pOrigin,173.93,73.21,0.00),v40,fine,tPen\WObj:=wPaper;
    MoveL Offs(pOrigin,173.93,73.21,6.00),v60,z5,tPen\WObj:=wPaper;
    MoveL Offs(pOrigin,174.99,74.28,6.00),vTravel,z5,tPen\WObj:=wPaper;
    MoveL Offs(pOrigin,174.99,74.28,0.00),v60,z0,tPen\WObj:=wPaper;
    MoveL Offs(pOrigin,175.62,74.91,0.00),v40,z0,tPen\WObj:=wPaper;
    MoveL Offs(pOrigin,174.99,74.28,0.00),v40,fine,tPen\WObj:=wPaper;
    MoveL Offs(pOrigin,174.99,74.28,6.00),v60,z5,tPen\WObj:=wPaper;
    MoveL Offs(pOrigin,174.77,75.97,6.00),vTravel,z5,tPen\WObj:=wPaper;
    MoveL Offs(pOrigin,174.77,75.97,0.00),v60,z0,tPen\WObj:=wPaper;
    MoveL Offs(pOrigin,175.20,76.40,0.00),v40,z0,tPen\WObj:=wPaper;
    MoveL Offs(pOrigin,174.77,75.97,0.00),v40,fine,tPen\WObj:=wPaper;
    MoveL Offs(pOrigin,174.77,75.97,6.00),v60,z5,tPen\WObj:=wPaper;
    MoveL Offs(pOrigin,172.65,71.94,6.00),vTravel,z5,tPen\WObj:=wPaper;
    MoveL Offs(pOrigin,172.65,71.94,0.00),v60,z0,tPen\WObj:=wPaper;
    MoveL Offs(pOrigin,173.71,73.00,0.00),v40,z0,tPen\WObj:=wPaper;
    MoveL Offs(pOrigin,172.65,71.94,0.00),v40,fine,tPen\WObj:=wPaper;
    MoveL Offs(pOrigin,172.65,71.94,6.00),v60,z5,tPen\WObj:=wPaper;
    MoveL Offs(pOrigin,169.25,68.96,6.00),vTravel,z5,tPen\WObj:=wPaper;
    MoveL Offs(pOrigin,169.25,68.96,0.00),v60,z0,tPen\WObj:=wPaper;
    MoveL Offs(pOrigin,169.68,69.39,0.00),v40,z0,tPen\WObj:=wPaper;
    MoveL Offs(pOrigin,169.25,68.96,0.00),v40,fine,tPen\WObj:=wPaper;
    MoveL Offs(pOrigin,169.25,68.96,6.00),v60,z5,tPen\WObj:=wPaper;
    MoveL Offs(pOrigin,181.57,66.20,6.00),vTravel,z5,tPen\WObj:=wPaper;
    MoveL Offs(pOrigin,181.57,66.20,0.00),v60,z0,tPen\WObj:=wPaper;
    MoveL Offs(pOrigin,182.85,64.71,0.00),v40,z0,tPen\WObj:=wPaper;
    MoveL Offs(pOrigin,184.34,63.86,0.00),v40,z0,tPen\WObj:=wPaper;
    MoveL Offs(pOrigin,183.91,64.07,0.00),v40,z0,tPen\WObj:=wPaper;
    MoveL Offs(pOrigin,184.34,63.86,0.00),v40,z0,tPen\WObj:=wPaper;
    MoveL Offs(pOrigin,183.91,64.07,0.00),v40,fine,tPen\WObj:=wPaper;
    MoveL Offs(pOrigin,183.91,64.07,6.00),v60,z5,tPen\WObj:=wPaper;
    MoveL Offs(pOrigin,181.15,52.39,6.00),vTravel,z5,tPen\WObj:=wPaper;
    MoveL Offs(pOrigin,181.15,52.39,0.00),v60,z0,tPen\WObj:=wPaper;
    MoveL Offs(pOrigin,183.70,50.90,0.00),v40,fine,tPen\WObj:=wPaper;
    MoveL Offs(pOrigin,183.70,50.90,6.00),v60,z5,tPen\WObj:=wPaper;
    MoveL Offs(pOrigin,200.49,33.26,6.00),vTravel,z5,tPen\WObj:=wPaper;
    MoveL Offs(pOrigin,200.49,33.26,0.00),v60,z0,tPen\WObj:=wPaper;
    MoveL Offs(pOrigin,201.34,34.75,0.00),v40,z0,tPen\WObj:=wPaper;
    MoveL Offs(pOrigin,202.61,35.39,0.00),v40,fine,tPen\WObj:=wPaper;
    MoveL Offs(pOrigin,202.61,35.39,6.00),v60,z5,tPen\WObj:=wPaper;
    MoveL Offs(pOrigin,205.59,37.51,6.00),vTravel,z5,tPen\WObj:=wPaper;
    MoveL Offs(pOrigin,205.59,37.51,0.00),v60,z0,tPen\WObj:=wPaper;
    MoveL Offs(pOrigin,206.01,37.72,0.00),v40,z0,tPen\WObj:=wPaper;
    MoveL Offs(pOrigin,205.59,37.51,0.00),v40,z0,tPen\WObj:=wPaper;
  ENDPROC

